LIN {X 0,Y 524.028,Z 204.208,A -85,B 0,C 180,E1 -4854.613,E2 -4854.613} C_VEL
LIN {X 0,Y 524.052,Z 204.202,A -85,B 0,C 180,E1 -4857.694,E2 -4857.694} C_VEL
LIN {X 0,Y 524.073,Z 204.206,A -85,B 0,C 180,E1 -4860.768,E2 -4860.768} C_VEL
LIN {X 0,Y 524.024,Z 204.211,A -85,B 0,C 180,E1 -4863.075,E2 -4863.075} C_VEL
LIN {X 0,Y 523.997,Z 204.21,A -85,B 0,C 180,E1 -4866.159,E2 -4866.159} C_VEL
LIN {X 0,Y 523.954,Z 204.219,A -85,B 0,C 180,E1 -4868.485,E2 -4868.485} C_VEL
LIN {X 0,Y 523.97,Z 204.212,A -85,B 0,C 180,E1 -4871.752,E2 -4871.752} C_VEL
LIN {X 0,Y 523.939,Z 204.219,A -85,B 0,C 180,E1 -4875.054,E2 -4875.054} C_VEL
LIN {X 0,Y 523.919,Z 204.219,A -85,B 0,C 180,E1 -4877.97,E2 -4877.97} C_VEL
LIN {X 0,Y 523.945,Z 204.222,A -85,B 0,C 180,E1 -4880.411,E2 -4880.411} C_VEL
LIN {X 0,Y 523.927,Z 204.221,A -85,B 0,C 180,E1 -4882.893,E2 -4882.893} C_VEL
LIN {X 0,Y 523.911,Z 204.219,A -85,B 0,C 180,E1 -4885.421,E2 -4885.421} C_VEL
LIN {X 0,Y 523.927,Z 204.221,A -85,B 0,C 180,E1 -4888.001,E2 -4888.001} C_VEL
LIN {X 0,Y 523.908,Z 204.222,A -85,B 0,C 180,E1 -4890.859,E2 -4890.859} C_VEL
LIN {X 0,Y 523.922,Z 204.22,A -85,B 0,C 180,E1 -4893.738,E2 -4893.738} C_VEL
LIN {X 0,Y 523.886,Z 204.229,A -85,B 0,C 180,E1 -4896.407,E2 -4896.407} C_VEL
LIN {X 0,Y 523.932,Z 204.217,A -85,B 0,C 180,E1 -4899.083,E2 -4899.083} C_VEL
LIN {X 0,Y 523.949,Z 204.215,A -85,B 0,C 180,E1 -4901.317,E2 -4901.317} C_VEL
LIN {X 0,Y 523.924,Z 204.219,A -85,B 0,C 180,E1 -4904.694,E2 -4904.694} C_VEL
LIN {X 0,Y 523.889,Z 204.222,A -85,B 0,C 180,E1 -4906.958,E2 -4906.958} C_VEL
LIN {X 0,Y 523.23,Z 204.308,A -85,B 0,C 180,E1 -4907.6,E2 -4907.6} C_VEL
LIN {X 0,Y 520.401,Z 204.663,A -85,B 0,C 180,E1 -4908.642,E2 -4908.642} C_VEL
LIN {X 0,Y 518.002,Z 204.964,A -85,B 0,C 180,E1 -4909.482,E2 -4909.482} C_VEL
LIN {X 0,Y 516.964,Z 205.091,A -85,B 0,C 180,E1 -4910.13,E2 -4910.13} C_VEL
LIN {X 0,Y 516.875,Z 205.099,A -85,B 0,C 180,E1 -4910.349,E2 -4910.349} C_VEL
LIN {X 0,Y 516.863,Z 205.099,A -85,B 0,C 180,E1 -4913.345,E2 -4913.345} C_VEL
LIN {X 0,Y 516.894,Z 205.098,A -85,B 0,C 180,E1 -4916.124,E2 -4916.124} C_VEL
LIN {X 0,Y 516.878,Z 205.095,A -85,B 0,C 180,E1 -4918.938,E2 -4918.938} C_VEL
LIN {X 0,Y 516.907,Z 205.098,A -85,B 0,C 180,E1 -4921.588,E2 -4921.588} C_VEL
LIN {X 0,Y 516.921,Z 205.092,A -85,B 0,C 180,E1 -4924.214,E2 -4924.214} C_VEL
LIN {X 0,Y 516.862,Z 205.097,A -85,B 0,C 180,E1 -4926.779,E2 -4926.779} C_VEL
LIN {X 0,Y 516.931,Z 205.096,A -85,B 0,C 180,E1 -4929.734,E2 -4929.734} C_VEL
LIN {X 0,Y 516.923,Z 205.09,A -85,B 0,C 180,E1 -4932.598,E2 -4932.598} C_VEL
LIN {X 0,Y 516.946,Z 205.09,A -85,B 0,C 180,E1 -4935.032,E2 -4935.032} C_VEL
LIN {X 0,Y 516.962,Z 205.085,A -85,B 0,C 180,E1 -4938.235,E2 -4938.235} C_VEL
LIN {X 0,Y 516.967,Z 205.093,A -85,B 0,C 180,E1 -4941.401,E2 -4941.401} C_VEL
LIN {X 0,Y 517,Z 205.083,A -85,B 0,C 180,E1 -4943.757,E2 -4943.757} C_VEL
LIN {X 0,Y 517.01,Z 205.082,A -85,B 0,C 180,E1 -4946.883,E2 -4946.883} C_VEL
LIN {X 0,Y 517.085,Z 205.07,A -85,B 0,C 180,E1 -4950,E2 -4950} C_VEL
LIN {X 0,Y 517.012,Z 205.088,A -85,B 0,C 180,E1 -4953.117,E2 -4953.117} C_VEL
LIN {X 0,Y 516.996,Z 205.081,A -85,B 0,C 180,E1 -4956.243,E2 -4956.243} C_VEL
LIN {X 0,Y 516.95,Z 205.09,A -85,B 0,C 180,E1 -4959.388,E2 -4959.388} C_VEL
LIN {X 0,Y 516.949,Z 205.087,A -85,B 0,C 180,E1 -4961.806,E2 -4961.806} C_VEL
LIN {X 0,Y 516.94,Z 205.093,A -85,B 0,C 180,E1 -4965.145,E2 -4965.145} C_VEL
LIN {X 0,Y 516.919,Z 205.091,A -85,B 0,C 180,E1 -4968.22,E2 -4968.22} C_VEL
LIN {X 0,Y 516.905,Z 205.099,A -85,B 0,C 180,E1 -4970.699,E2 -4970.699} C_VEL
LIN {X 0,Y 516.901,Z 205.093,A -85,B 0,C 180,E1 -4974.07,E2 -4974.07} C_VEL
LIN {X 0,Y 516.917,Z 205.1,A -85,B 0,C 180,E1 -4976.655,E2 -4976.655} C_VEL
LIN {X 0,Y 516.913,Z 205.095,A -85,B 0,C 180,E1 -4979.525,E2 -4979.525} C_VEL
LIN {X 0,Y 516.991,Z 205.141,A -85,B 0,C 180,E1 -4980.941,E2 -4980.941} C_VEL
LIN {X 0,Y 517.439,Z 210.279,A -85,B 0,C 180,E1 -4981.982,E2 -4981.982} C_VEL
LIN {X 0,Y 517.248,Z 224.094,A -85,B 0,C 180,E1 -4984.686,E2 -4984.686} C_VEL
LIN {X 0,Y 519.109,Z 235.104,A -85,B 0,C 180,E1 -4984.919,E2 -4984.919} C_VEL
LIN {X 0,Y 518.527,Z 331.623,A -85,B 0,C 180,E1 -4986.303,E2 -4986.303} C_VEL
LIN {X 0,Y 518.327,Z 345.145,A -85,B 0,C 180,E1 -4986.668,E2 -4986.668} C_VEL
LIN {X 0,Y 518.194,Z 357.087,A -85,B 0,C 180,E1 -4987.144,E2 -4987.144} C_VEL
LIN {X 0,Y 517.927,Z 368.274,A -85,B 0,C 180,E1 -4987.737,E2 -4987.737} C_VEL
LIN {X 0,Y 517.619,Z 379.34,A -85,B 0,C 180,E1 -4988.487,E2 -4988.487} C_VEL
LIN {X 0,Y 517.308,Z 390.499,A -85,B 0,C 180,E1 -4989.437,E2 -4989.437} C_VEL
LIN {X 0,Y 517.044,Z 399.867,A -85,B 0,C 180,E1 -4990.431,E2 -4990.431} C_VEL
LIN {X 0,Y 516.822,Z 408.68,A -85,B 0,C 180,E1 -4991.59,E2 -4991.59} C_VEL
LIN {X 0,Y 516.577,Z 416.392,A -85,B 0,C 180,E1 -4992.857,E2 -4992.857} C_VEL
LIN {X 0,Y 516.485,Z 422.702,A -85,B 0,C 180,E1 -4994.189,E2 -4994.189} C_VEL
LIN {X 0,Y 516.339,Z 427.576,A -85,B 0,C 180,E1 -4995.541,E2 -4995.541} C_VEL
LIN {X 0,Y 516.293,Z 430.487,A -85,B 0,C 180,E1 -4996.636,E2 -4996.636} C_VEL
LIN {X 0,Y 516.24,Z 433.161,A -85,B 0,C 180,E1 -4998.159,E2 -4998.159} C_VEL
LIN {X 0,Y 516.175,Z 434.262,A -85,B 0,C 180,E1 -4999.675,E2 -4999.675} C_VEL
LIN {X 0,Y 516.192,Z 433.883,A -85,B 0,C 180,E1 -5001.223,E2 -5001.223} C_VEL
LIN {X 0,Y 516.191,Z 432.79,A -85,B 0,C 180,E1 -5002.217,E2 -5002.217} C_VEL
LIN {X 0,Y 516.28,Z 430.595,A -85,B 0,C 180,E1 -5003.424,E2 -5003.424} C_VEL
LIN {X 0,Y 516.358,Z 427.029,A -85,B 0,C 180,E1 -5004.741,E2 -5004.741} C_VEL
LIN {X 0,Y 516.425,Z 421.942,A -85,B 0,C 180,E1 -5006.104,E2 -5006.104} C_VEL
LIN {X 0,Y 516.6,Z 416.145,A -85,B 0,C 180,E1 -5007.295,E2 -5007.295} C_VEL
LIN {X 0,Y 516.793,Z 409.28,A -85,B 0,C 180,E1 -5008.428,E2 -5008.428} C_VEL
LIN {X 0,Y 517.047,Z 400.626,A -85,B 0,C 180,E1 -5009.581,E2 -5009.581} C_VEL
LIN {X 0,Y 517.308,Z 391.616,A -85,B 0,C 180,E1 -5010.557,E2 -5010.557} C_VEL
LIN {X 0,Y 517.528,Z 382.117,A -85,B 0,C 180,E1 -5011.4,E2 -5011.4} C_VEL
LIN {X 0,Y 517.83,Z 371.744,A -85,B 0,C 180,E1 -5012.145,E2 -5012.145} C_VEL
LIN {X 0,Y 518.169,Z 359.936,A -85,B 0,C 180,E1 -5012.813,E2 -5012.813} C_VEL
LIN {X 0,Y 518.374,Z 348.271,A -85,B 0,C 180,E1 -5013.314,E2 -5013.314} C_VEL
LIN {X 0,Y 518.512,Z 335.514,A -85,B 0,C 180,E1 -5013.702,E2 -5013.702} C_VEL
LIN {X 0,Y 518.61,Z 319.67,A -85,B 0,C 180,E1 -5013.977,E2 -5013.977} C_VEL
LIN {X 0,Y 519.05,Z 233.514,A -85,B 0,C 180,E1 -5015.201,E2 -5015.201} C_VEL
LIN {X 0,Y 517.236,Z 223.957,A -85,B 0,C 180,E1 -5015.41,E2 -5015.41} C_VEL
LIN {X 0,Y 517.224,Z 207.844,A -85,B 0,C 180,E1 -5018.268,E2 -5018.268} C_VEL
LIN {X 0,Y 516.917,Z 205.098,A -85,B 0,C 180,E1 -5018.778,E2 -5018.778} C_VEL
LIN {X 0,Y 516.879,Z 205.098,A -85,B 0,C 180,E1 -5022.117,E2 -5022.117} C_VEL
LIN {X 0,Y 516.897,Z 205.1,A -85,B 0,C 180,E1 -5025.029,E2 -5025.029} C_VEL
LIN {X 0,Y 516.951,Z 205.09,A -85,B 0,C 180,E1 -5028.234,E2 -5028.234} C_VEL
LIN {X 0,Y 516.92,Z 205.098,A -85,B 0,C 180,E1 -5031.399,E2 -5031.399} C_VEL
LIN {X 0,Y 516.966,Z 205.088,A -85,B 0,C 180,E1 -5033.757,E2 -5033.757} C_VEL
LIN {X 0,Y 516.966,Z 205.091,A -85,B 0,C 180,E1 -5036.883,E2 -5036.883} C_VEL
LIN {X 0,Y 517.024,Z 205.079,A -85,B 0,C 180,E1 -5040,E2 -5040} C_VEL
LIN {X 0,Y 516.964,Z 205.092,A -85,B 0,C 180,E1 -5043.118,E2 -5043.118} C_VEL
LIN {X 0,Y 516.947,Z 205.087,A -85,B 0,C 180,E1 -5046.244,E2 -5046.244} C_VEL
LIN {X 0,Y 516.907,Z 205.095,A -85,B 0,C 180,E1 -5049.39,E2 -5049.39} C_VEL
LIN {X 0,Y 516.931,Z 205.088,A -85,B 0,C 180,E1 -5051.826,E2 -5051.826} C_VEL
LIN {X 0,Y 516.891,Z 205.098,A -85,B 0,C 180,E1 -5055.147,E2 -5055.147} C_VEL
LIN {X 0,Y 516.881,Z 205.097,A -85,B 0,C 180,E1 -5058.224,E2 -5058.224} C_VEL
LIN {X 0,Y 516.867,Z 205.104,A -85,B 0,C 180,E1 -5060.704,E2 -5060.704} C_VEL
LIN {X 0,Y 516.844,Z 205.099,A -85,B 0,C 180,E1 -5063.225,E2 -5063.225} C_VEL
LIN {X 0,Y 516.9,Z 205.097,A -85,B 0,C 180,E1 -5066.199,E2 -5066.199} C_VEL
LIN {X 0,Y 516.881,Z 205.094,A -85,B 0,C 180,E1 -5069.307,E2 -5069.307} C_VEL
LIN {X 0,Y 516.861,Z 205.104,A -85,B 0,C 180,E1 -5072.547,E2 -5072.547} C_VEL
LIN {X 0,Y 516.846,Z 205.098,A -85,B 0,C 180,E1 -5075.335,E2 -5075.335} C_VEL
LIN {X 0,Y 516.847,Z 205.103,A -85,B 0,C 180,E1 -5077.946,E2 -5077.946} C_VEL
LIN {X 0,Y 516.854,Z 205.101,A -85,B 0,C 180,E1 -5080.745,E2 -5080.745} C_VEL
LIN {X 0,Y 516.855,Z 205.099,A -85,B 0,C 180,E1 -5082.835,E2 -5082.835} C_VEL
LIN {X 0,Y 516.869,Z 205.097,A -85,B 0,C 180,E1 -5085.01,E2 -5085.01} C_VEL
LIN {X 0,Y 516.894,Z 205.099,A -85,B 0,C 180,E1 -5088.402,E2 -5088.402} C_VEL
LIN {X 0,Y 516.86,Z 205.099,A -85,B 0,C 180,E1 -5091.287,E2 -5091.287} C_VEL
LIN {X 0,Y 516.871,Z 205.103,A -85,B 0,C 180,E1 -5094.224,E2 -5094.224} C_VEL
LIN {X 0,Y 516.88,Z 205.097,A -85,B 0,C 180,E1 -5097.056,E2 -5097.056} C_VEL
LIN {X 0,Y 516.88,Z 205.104,A -85,B 0,C 180,E1 -5099.799,E2 -5099.799} C_VEL
LIN {X 0,Y 516.915,Z 205.096,A -85,B 0,C 180,E1 -5102.47,E2 -5102.47} C_VEL
LIN {X 0,Y 516.957,Z 205.158,A -85,B 0,C 180,E1 -5105.114,E2 -5105.114} C_VEL
LIN {X 0,Y 518.311,Z 213.375,A -85,B 0,C 180,E1 -5106.424,E2 -5106.424} C_VEL
LIN {X 0,Y 517.948,Z 232.817,A -85,B 0,C 180,E1 -5109.344,E2 -5109.344} C_VEL
LIN {X 0,Y 517.523,Z 253.595,A -85,B 0,C 180,E1 -5112.442,E2 -5112.442} C_VEL
LIN {X 0,Y 517.213,Z 268.372,A -85,B 0,C 180,E1 -5114.627,E2 -5114.627} C_VEL
LIN {X 0,Y 519.009,Z 281.849,A -85,B 0,C 180,E1 -5114.879,E2 -5114.879} C_VEL
LIN {X 0,Y 518.499,Z 377.861,A -85,B 0,C 180,E1 -5116.255,E2 -5116.255} C_VEL
LIN {X 0,Y 518.253,Z 391.659,A -85,B 0,C 180,E1 -5116.623,E2 -5116.623} C_VEL
LIN {X 0,Y 517.973,Z 404.074,A -85,B 0,C 180,E1 -5117.114,E2 -5117.114} C_VEL
LIN {X 0,Y 517.695,Z 416.837,A -85,B 0,C 180,E1 -5117.808,E2 -5117.808} C_VEL
LIN {X 0,Y 517.391,Z 428.749,A -85,B 0,C 180,E1 -5118.642,E2 -5118.642} C_VEL
LIN {X 0,Y 517.132,Z 437.799,A -85,B 0,C 180,E1 -5119.429,E2 -5119.429} C_VEL
LIN {X 0,Y 516.852,Z 447.086,A -85,B 0,C 180,E1 -5120.412,E2 -5120.412} C_VEL
LIN {X 0,Y 516.635,Z 456.126,A -85,B 0,C 180,E1 -5121.592,E2 -5121.592} C_VEL
LIN {X 0,Y 516.502,Z 463.409,A -85,B 0,C 180,E1 -5122.77,E2 -5122.77} C_VEL
LIN {X 0,Y 516.383,Z 468.318,A -85,B 0,C 180,E1 -5123.75,E2 -5123.75} C_VEL
LIN {X 0,Y 516.312,Z 473.094,A -85,B 0,C 180,E1 -5124.924,E2 -5124.924} C_VEL
LIN {X 0,Y 516.37,Z 476.747,A -85,B 0,C 180,E1 -5126.098,E2 -5126.098} C_VEL
LIN {X 0,Y 516.282,Z 478.629,A -85,B 0,C 180,E1 -5126.879,E2 -5126.879} C_VEL
LIN {X 0,Y 516.261,Z 480.041,A -85,B 0,C 180,E1 -5127.66,E2 -5127.66} C_VEL
LIN {X 0,Y 516.167,Z 481.664,A -85,B 0,C 180,E1 -5129.22,E2 -5129.22} C_VEL
LIN {X 0,Y 516.167,Z 481.887,A -85,B 0,C 180,E1 -5130,E2 -5130} C_VEL
LIN {X 0,Y 516.192,Z 481.066,A -85,B 0,C 180,E1 -5131.56,E2 -5131.56} C_VEL
LIN {X 0,Y 516.261,Z 480.07,A -85,B 0,C 180,E1 -5132.34,E2 -5132.34} C_VEL
LIN {X 0,Y 516.282,Z 478.667,A -85,B 0,C 180,E1 -5133.121,E2 -5133.121} C_VEL
LIN {X 0,Y 516.311,Z 475.715,A -85,B 0,C 180,E1 -5134.293,E2 -5134.293} C_VEL
LIN {X 0,Y 516.368,Z 471.715,A -85,B 0,C 180,E1 -5135.466,E2 -5135.466} C_VEL
LIN {X 0,Y 516.439,Z 465.782,A -85,B 0,C 180,E1 -5136.794,E2 -5136.794} C_VEL
LIN {X 0,Y 516.592,Z 458.83,A -85,B 0,C 180,E1 -5138.015,E2 -5138.015} C_VEL
LIN {X 0,Y 516.77,Z 450.482,A -85,B 0,C 180,E1 -5139.194,E2 -5139.194} C_VEL
LIN {X 0,Y 516.971,Z 441.909,A -85,B 0,C 180,E1 -5140.178,E2 -5140.178} C_VEL
LIN {X 0,Y 517.33,Z 431.327,A -85,B 0,C 180,E1 -5141.161,E2 -5141.161} C_VEL
LIN {X 0,Y 517.674,Z 420.056,A -85,B 0,C 180,E1 -5142.002,E2 -5142.002} C_VEL
LIN {X 0,Y 517.9,Z 409.336,A -85,B 0,C 180,E1 -5142.638,E2 -5142.638} C_VEL
LIN {X 0,Y 518.141,Z 397.418,A -85,B 0,C 180,E1 -5143.18,E2 -5143.18} C_VEL
LIN {X 0,Y 518.418,Z 383.678,A -85,B 0,C 180,E1 -5143.622,E2 -5143.622} C_VEL
LIN {X 0,Y 518.627,Z 371.26,A -85,B 0,C 180,E1 -5143.866,E2 -5143.866} C_VEL
LIN {X 0,Y 518.844,Z 279.698,A -85,B 0,C 180,E1 -5145.162,E2 -5145.162} C_VEL
LIN {X 0,Y 517.252,Z 268.853,A -85,B 0,C 180,E1 -5145.371,E2 -5145.371} C_VEL
LIN {X 0,Y 517.694,Z 248.791,A -85,B 0,C 180,E1 -5148.397,E2 -5148.397} C_VEL
LIN {X 0,Y 518.264,Z 228.616,A -85,B 0,C 180,E1 -5151.475,E2 -5151.475} C_VEL
LIN {X 0,Y 518.602,Z 213.817,A -85,B 0,C 180,E1 -5153.773,E2 -5153.773} C_VEL
LIN {X 0,Y 516.949,Z 205.092,A -85,B 0,C 180,E1 -5155.246,E2 -5155.246} C_VEL
LIN {X 0,Y 516.904,Z 205.099,A -85,B 0,C 180,E1 -5158.413,E2 -5158.413} C_VEL
LIN {X 0,Y 516.876,Z 205.097,A -85,B 0,C 180,E1 -5161.106,E2 -5161.106} C_VEL
LIN {X 0,Y 516.895,Z 205.102,A -85,B 0,C 180,E1 -5163.963,E2 -5163.963} C_VEL
LIN {X 0,Y 516.864,Z 205.097,A -85,B 0,C 180,E1 -5166.742,E2 -5166.742} C_VEL
LIN {X 0,Y 516.86,Z 205.104,A -85,B 0,C 180,E1 -5169.718,E2 -5169.718} C_VEL
LIN {X 0,Y 516.891,Z 205.102,A -85,B 0,C 180,E1 -5171.771,E2 -5171.771} C_VEL
LIN {X 0,Y 516.896,Z 205.093,A -85,B 0,C 180,E1 -5175.007,E2 -5175.007} C_VEL
LIN {X 0,Y 516.886,Z 205.095,A -85,B 0,C 180,E1 -5178.395,E2 -5178.395} C_VEL
LIN {X 0,Y 516.847,Z 205.103,A -85,B 0,C 180,E1 -5181.281,E2 -5181.281} C_VEL
LIN {X 0,Y 516.855,Z 205.1,A -85,B 0,C 180,E1 -5184.218,E2 -5184.218} C_VEL
LIN {X 0,Y 516.859,Z 205.1,A -85,B 0,C 180,E1 -5187.05,E2 -5187.05} C_VEL
LIN {X 0,Y 516.85,Z 205.104,A -85,B 0,C 180,E1 -5189.793,E2 -5189.793} C_VEL
LIN {X 0,Y 516.886,Z 205.094,A -85,B 0,C 180,E1 -5192.465,E2 -5192.465} C_VEL
LIN {X 0,Y 516.867,Z 205.101,A -85,B 0,C 180,E1 -5195.069,E2 -5195.069} C_VEL
LIN {X 0,Y 516.866,Z 205.102,A -85,B 0,C 180,E1 -5197.621,E2 -5197.621} C_VEL
LIN {X 0,Y 516.883,Z 205.095,A -85,B 0,C 180,E1 -5200.128,E2 -5200.128} C_VEL
LIN {X 0,Y 516.891,Z 205.095,A -85,B 0,C 180,E1 -5202.595,E2 -5202.595} C_VEL
LIN {X 0,Y 516.888,Z 205.1,A -85,B 0,C 180,E1 -5205.028,E2 -5205.028} C_VEL
LIN {X 0,Y 516.951,Z 205.086,A -85,B 0,C 180,E1 -5208.233,E2 -5208.233} C_VEL
LIN {X 0,Y 516.917,Z 205.095,A -85,B 0,C 180,E1 -5211.399,E2 -5211.399} C_VEL
LIN {X 0,Y 516.946,Z 205.088,A -85,B 0,C 180,E1 -5213.756,E2 -5213.756} C_VEL
LIN {X 0,Y 516.963,Z 205.092,A -85,B 0,C 180,E1 -5216.882,E2 -5216.882} C_VEL
LIN {X 0,Y 517.023,Z 205.077,A -85,B 0,C 180,E1 -5220,E2 -5220} C_VEL
LIN {X 0,Y 516.965,Z 205.09,A -85,B 0,C 180,E1 -5223.117,E2 -5223.117} C_VEL
LIN {X 0,Y 516.965,Z 205.086,A -85,B 0,C 180,E1 -5226.243,E2 -5226.243} C_VEL
LIN {X 0,Y 516.919,Z 205.097,A -85,B 0,C 180,E1 -5228.601,E2 -5228.601} C_VEL
LIN {X 0,Y 516.929,Z 205.089,A -85,B 0,C 180,E1 -5231.825,E2 -5231.825} C_VEL
LIN {X 0,Y 516.892,Z 205.096,A -85,B 0,C 180,E1 -5235.148,E2 -5235.148} C_VEL
LIN {X 0,Y 516.879,Z 205.099,A -85,B 0,C 180,E1 -5238.224,E2 -5238.224} C_VEL
LIN {X 0,Y 516.884,Z 205.101,A -85,B 0,C 180,E1 -5240.702,E2 -5240.702} C_VEL
LIN {X 0,Y 516.867,Z 205.097,A -85,B 0,C 180,E1 -5243.223,E2 -5243.223} C_VEL
LIN {X 0,Y 516.898,Z 205.098,A -85,B 0,C 180,E1 -5246.199,E2 -5246.199} C_VEL
LIN {X 0,Y 516.898,Z 205.093,A -85,B 0,C 180,E1 -5249.306,E2 -5249.306} C_VEL
LIN {X 0,Y 516.859,Z 205.103,A -85,B 0,C 180,E1 -5252.547,E2 -5252.547} C_VEL
LIN {X 0,Y 516.844,Z 205.1,A -85,B 0,C 180,E1 -5255.335,E2 -5255.335} C_VEL
LIN {X 0,Y 516.846,Z 205.104,A -85,B 0,C 180,E1 -5257.946,E2 -5257.946} C_VEL
LIN {X 0,Y 516.883,Z 205.096,A -85,B 0,C 180,E1 -5260.741,E2 -5260.741} C_VEL
LIN {X 0,Y 516.851,Z 205.105,A -85,B 0,C 180,E1 -5263.906,E2 -5263.906} C_VEL
LIN {X 0,Y 516.853,Z 205.107,A -85,B 0,C 180,E1 -5266.11,E2 -5266.11} C_VEL
LIN {X 0,Y 516.886,Z 205.095,A -85,B 0,C 180,E1 -5269.264,E2 -5269.264} C_VEL
LIN {X 0,Y 516.875,Z 205.099,A -85,B 0,C 180,E1 -5270.349,E2 -5270.349} C_VEL
LIN {X 0,Y 516.197,Z 205.181,A -85,B 0,C 180,E1 -5270.999,E2 -5270.999} C_VEL
LIN {X 0,Y 513.342,Z 205.543,A -85,B 0,C 180,E1 -5272.055,E2 -5272.055} C_VEL
LIN {X 0,Y 510.933,Z 205.845,A -85,B 0,C 180,E1 -5272.905,E2 -5272.905} C_VEL
LIN {X 0,Y 509.895,Z 205.971,A -85,B 0,C 180,E1 -5273.562,E2 -5273.562} C_VEL
LIN {X 0,Y 509.808,Z 205.98,A -85,B 0,C 180,E1 -5273.784,E2 -5273.784} C_VEL
LIN {X 0,Y 509.845,Z 205.972,A -85,B 0,C 180,E1 -5276.542,E2 -5276.542} C_VEL
LIN {X 0,Y 509.834,Z 205.976,A -85,B 0,C 180,E1 -5279.337,E2 -5279.337} C_VEL
LIN {X 0,Y 509.881,Z 205.971,A -85,B 0,C 180,E1 -5282.057,E2 -5282.057} C_VEL
LIN {X 0,Y 509.867,Z 205.969,A -85,B 0,C 180,E1 -5284.707,E2 -5284.707} C_VEL
LIN {X 0,Y 509.827,Z 205.98,A -85,B 0,C 180,E1 -5287.457,E2 -5287.457} C_VEL
LIN {X 0,Y 509.909,Z 205.969,A -85,B 0,C 180,E1 -5289.847,E2 -5289.847} C_VEL
LIN {X 0,Y 509.879,Z 205.971,A -85,B 0,C 180,E1 -5293.177,E2 -5293.177} C_VEL
LIN {X 0,Y 509.868,Z 205.975,A -85,B 0,C 180,E1 -5295.636,E2 -5295.636} C_VEL
LIN {X 0,Y 509.91,Z 205.965,A -85,B 0,C 180,E1 -5298.876,E2 -5298.876} C_VEL
LIN {X 0,Y 509.949,Z 205.959,A -85,B 0,C 180,E1 -5302.079,E2 -5302.079} C_VEL
LIN {X 0,Y 509.978,Z 205.955,A -85,B 0,C 180,E1 -5304.465,E2 -5304.465} C_VEL
LIN {X 0,Y 510.055,Z 205.949,A -85,B 0,C 180,E1 -5307.631,E2 -5307.631} C_VEL
LIN {X 0,Y 510.062,Z 205.948,A -85,B 0,C 180,E1 -5310.789,E2 -5310.789} C_VEL
LIN {X 0,Y 509.954,Z 205.967,A -85,B 0,C 180,E1 -5313.16,E2 -5313.16} C_VEL
LIN {X 0,Y 509.943,Z 205.96,A -85,B 0,C 180,E1 -5316.329,E2 -5316.329} C_VEL
LIN {X 0,Y 509.913,Z 205.967,A -85,B 0,C 180,E1 -5318.719,E2 -5318.719} C_VEL
LIN {X 0,Y 509.901,Z 205.964,A -85,B 0,C 180,E1 -5321.93,E2 -5321.93} C_VEL
LIN {X 0,Y 509.889,Z 205.97,A -85,B 0,C 180,E1 -5325.24,E2 -5325.24} C_VEL
LIN {X 0,Y 509.883,Z 205.967,A -85,B 0,C 180,E1 -5327.999,E2 -5327.999} C_VEL
LIN {X 0,Y 509.843,Z 205.978,A -85,B 0,C 180,E1 -5331,E2 -5331} C_VEL
LIN {X 0,Y 509.827,Z 205.974,A -85,B 0,C 180,E1 -5333.561,E2 -5333.561} C_VEL
LIN {X 0,Y 509.902,Z 205.97,A -85,B 0,C 180,E1 -5336.377,E2 -5336.377} C_VEL
LIN {X 0,Y 509.872,Z 205.976,A -85,B 0,C 180,E1 -5338.841,E2 -5338.841} C_VEL
LIN {X 0,Y 509.958,Z 205.983,A -85,B 0,C 180,E1 -5340.81,E2 -5340.81} C_VEL
LIN {X 0,Y 510.45,Z 210.705,A -85,B 0,C 180,E1 -5341.775,E2 -5341.775} C_VEL
LIN {X 0,Y 510.23,Z 224.338,A -85,B 0,C 180,E1 -5344.47,E2 -5344.47} C_VEL
LIN {X 0,Y 512.23,Z 234.881,A -85,B 0,C 180,E1 -5344.704,E2 -5344.704} C_VEL
LIN {X 0,Y 511.675,Z 330.813,A -85,B 0,C 180,E1 -5346.097,E2 -5346.097} C_VEL
LIN {X 0,Y 511.437,Z 344.08,A -85,B 0,C 180,E1 -5346.445,E2 -5346.445} C_VEL
LIN {X 0,Y 511.286,Z 357.191,A -85,B 0,C 180,E1 -5346.964,E2 -5346.964} C_VEL
LIN {X 0,Y 510.973,Z 369.148,A -85,B 0,C 180,E1 -5347.609,E2 -5347.609} C_VEL
LIN {X 0,Y 510.631,Z 380.814,A -85,B 0,C 180,E1 -5348.424,E2 -5348.424} C_VEL
LIN {X 0,Y 510.313,Z 390.903,A -85,B 0,C 180,E1 -5349.304,E2 -5349.304} C_VEL
LIN {X 0,Y 510.028,Z 400.624,A -85,B 0,C 180,E1 -5350.359,E2 -5350.359} C_VEL
LIN {X 0,Y 509.805,Z 408.629,A -85,B 0,C 180,E1 -5351.425,E2 -5351.425} C_VEL
LIN {X 0,Y 509.538,Z 415.352,A -85,B 0,C 180,E1 -5352.514,E2 -5352.514} C_VEL
LIN {X 0,Y 509.406,Z 422.088,A -85,B 0,C 180,E1 -5353.885,E2 -5353.885} C_VEL
LIN {X 0,Y 509.291,Z 427.23,A -85,B 0,C 180,E1 -5355.27,E2 -5355.27} C_VEL
LIN {X 0,Y 509.234,Z 430.296,A -85,B 0,C 180,E1 -5356.366,E2 -5356.366} C_VEL
LIN {X 0,Y 509.164,Z 432.48,A -85,B 0,C 180,E1 -5357.442,E2 -5357.442} C_VEL
LIN {X 0,Y 509.146,Z 433.872,A -85,B 0,C 180,E1 -5358.504,E2 -5358.504} C_VEL
LIN {X 0,Y 509.105,Z 434.56,A -85,B 0,C 180,E1 -5359.548,E2 -5359.548} C_VEL
LIN {X 0,Y 509.129,Z 434.553,A -85,B 0,C 180,E1 -5360.618,E2 -5360.618} C_VEL
LIN {X 0,Y 509.098,Z 433.597,A -85,B 0,C 180,E1 -5361.886,E2 -5361.886} C_VEL
LIN {X 0,Y 509.169,Z 431.562,A -85,B 0,C 180,E1 -5363.176,E2 -5363.176} C_VEL
LIN {X 0,Y 509.267,Z 428.061,A -85,B 0,C 180,E1 -5364.577,E2 -5364.577} C_VEL
LIN {X 0,Y 509.333,Z 423.536,A -85,B 0,C 180,E1 -5365.875,E2 -5365.875} C_VEL
LIN {X 0,Y 509.546,Z 417.111,A -85,B 0,C 180,E1 -5367.273,E2 -5367.273} C_VEL
LIN {X 0,Y 509.738,Z 410.51,A -85,B 0,C 180,E1 -5368.404,E2 -5368.404} C_VEL
LIN {X 0,Y 510.004,Z 402.045,A -85,B 0,C 180,E1 -5369.574,E2 -5369.574} C_VEL
LIN {X 0,Y 510.314,Z 392.712,A -85,B 0,C 180,E1 -5370.619,E2 -5370.619} C_VEL
LIN {X 0,Y 510.566,Z 383.025,A -85,B 0,C 180,E1 -5371.504,E2 -5371.504} C_VEL
LIN {X 0,Y 510.909,Z 371.564,A -85,B 0,C 180,E1 -5372.338,E2 -5372.338} C_VEL
LIN {X 0,Y 511.224,Z 359.501,A -85,B 0,C 180,E1 -5373.021,E2 -5373.021} C_VEL
LIN {X 0,Y 511.493,Z 346.514,A -85,B 0,C 180,E1 -5373.566,E2 -5373.566} C_VEL
LIN {X 0,Y 511.642,Z 333.326,A -85,B 0,C 180,E1 -5373.938,E2 -5373.938} C_VEL
LIN {X 0,Y 511.818,Z 308.174,A -85,B 0,C 180,E1 -5374.331,E2 -5374.331} C_VEL
LIN {X 0,Y 512.249,Z 234.752,A -85,B 0,C 180,E1 -5375.393,E2 -5375.393} C_VEL
LIN {X 0,Y 510.249,Z 224.241,A -85,B 0,C 180,E1 -5375.621,E2 -5375.621} C_VEL
LIN {X 0,Y 510.235,Z 208.761,A -85,B 0,C 180,E1 -5378.38,E2 -5378.38} C_VEL
LIN {X 0,Y 509.881,Z 205.975,A -85,B 0,C 180,E1 -5378.894,E2 -5378.894} C_VEL
LIN {X 0,Y 509.858,Z 205.972,A -85,B 0,C 180,E1 -5382.347,E2 -5382.347} C_VEL
LIN {X 0,Y 509.824,Z 205.983,A -85,B 0,C 180,E1 -5385.633,E2 -5385.633} C_VEL
LIN {X 0,Y 509.891,Z 205.97,A -85,B 0,C 180,E1 -5388.1,E2 -5388.1} C_VEL
LIN {X 0,Y 509.867,Z 205.978,A -85,B 0,C 180,E1 -5391.279,E2 -5391.279} C_VEL
LIN {X 0,Y 509.937,Z 205.964,A -85,B 0,C 180,E1 -5393.67,E2 -5393.67} C_VEL
LIN {X 0,Y 509.908,Z 205.969,A -85,B 0,C 180,E1 -5396.84,E2 -5396.84} C_VEL
LIN {X 0,Y 510.014,Z 205.959,A -85,B 0,C 180,E1 -5399.211,E2 -5399.211} C_VEL
LIN {X 0,Y 509.882,Z 205.97,A -85,B 0,C 180,E1 -5401.58,E2 -5401.58} C_VEL
LIN {X 0,Y 509.906,Z 205.971,A -85,B 0,C 180,E1 -5403.161,E2 -5403.161} C_VEL
LIN {X 0,Y 509.898,Z 205.965,A -85,B 0,C 180,E1 -5406.331,E2 -5406.331} C_VEL
LIN {X 0,Y 509.865,Z 205.975,A -85,B 0,C 180,E1 -5408.721,E2 -5408.721} C_VEL
LIN {X 0,Y 509.9,Z 205.964,A -85,B 0,C 180,E1 -5411.932,E2 -5411.932} C_VEL
LIN {X 0,Y 509.844,Z 205.975,A -85,B 0,C 180,E1 -5415.244,E2 -5415.244} C_VEL
LIN {X 0,Y 509.84,Z 205.972,A -85,B 0,C 180,E1 -5418.003,E2 -5418.003} C_VEL
LIN {X 0,Y 509.809,Z 205.981,A -85,B 0,C 180,E1 -5421.004,E2 -5421.004} C_VEL
LIN {X 0,Y 509.804,Z 205.975,A -85,B 0,C 180,E1 -5423.565,E2 -5423.565} C_VEL
LIN {X 0,Y 509.869,Z 205.975,A -85,B 0,C 180,E1 -5426.381,E2 -5426.381} C_VEL
LIN {X 0,Y 509.836,Z 205.976,A -85,B 0,C 180,E1 -5428.847,E2 -5428.847} C_VEL
LIN {X 0,Y 509.785,Z 205.98,A -85,B 0,C 180,E1 -5431.593,E2 -5431.593} C_VEL
LIN {X 0,Y 509.816,Z 205.983,A -85,B 0,C 180,E1 -5434.416,E2 -5434.416} C_VEL
LIN {X 0,Y 509.785,Z 205.98,A -85,B 0,C 180,E1 -5437.344,E2 -5437.344} C_VEL
LIN {X 0,Y 509.807,Z 205.983,A -85,B 0,C 180,E1 -5440.386,E2 -5440.386} C_VEL
LIN {X 0,Y 509.795,Z 205.977,A -85,B 0,C 180,E1 -5443.066,E2 -5443.066} C_VEL
LIN {X 0,Y 509.797,Z 205.981,A -85,B 0,C 180,E1 -5445.797,E2 -5445.797} C_VEL
LIN {X 0,Y 509.836,Z 205.976,A -85,B 0,C 180,E1 -5448.578,E2 -5448.578} C_VEL
LIN {X 0,Y 509.831,Z 205.979,A -85,B 0,C 180,E1 -5451.79,E2 -5451.79} C_VEL
LIN {X 0,Y 509.827,Z 205.976,A -85,B 0,C 180,E1 -5454.626,E2 -5454.626} C_VEL
LIN {X 0,Y 509.847,Z 205.976,A -85,B 0,C 180,E1 -5457.484,E2 -5457.484} C_VEL
LIN {X 0,Y 509.848,Z 205.979,A -85,B 0,C 180,E1 -5460.277,E2 -5460.277} C_VEL
LIN {X 0,Y 509.873,Z 205.972,A -85,B 0,C 180,E1 -5462.947,E2 -5462.947} C_VEL
LIN {X 0,Y 509.909,Z 206.106,A -85,B 0,C 180,E1 -5464.963,E2 -5464.963} C_VEL
LIN {X 0,Y 511.329,Z 214.333,A -85,B 0,C 180,E1 -5466.298,E2 -5466.298} C_VEL
LIN {X 0,Y 511.005,Z 232.375,A -85,B 0,C 180,E1 -5469.05,E2 -5469.05} C_VEL
LIN {X 0,Y 510.502,Z 254.403,A -85,B 0,C 180,E1 -5472.372,E2 -5472.372} C_VEL
LIN {X 0,Y 510.216,Z 267.995,A -85,B 0,C 180,E1 -5474.409,E2 -5474.409} C_VEL
LIN {X 0,Y 512.149,Z 282.754,A -85,B 0,C 180,E1 -5474.69,E2 -5474.69} C_VEL
LIN {X 0,Y 511.617,Z 377.203,A -85,B 0,C 180,E1 -5476.066,E2 -5476.066} C_VEL
LIN {X 0,Y 511.331,Z 390.33,A -85,B 0,C 180,E1 -5476.413,E2 -5476.413} C_VEL
LIN {X 0,Y 511.033,Z 403.576,A -85,B 0,C 180,E1 -5476.936,E2 -5476.936} C_VEL
LIN {X 0,Y 510.753,Z 416.122,A -85,B 0,C 180,E1 -5477.623,E2 -5477.623} C_VEL
LIN {X 0,Y 510.396,Z 427.015,A -85,B 0,C 180,E1 -5478.383,E2 -5478.383} C_VEL
LIN {X 0,Y 510.126,Z 437.385,A -85,B 0,C 180,E1 -5479.282,E2 -5479.282} C_VEL
LIN {X 0,Y 509.82,Z 446.69,A -85,B 0,C 180,E1 -5480.279,E2 -5480.279} C_VEL
LIN {X 0,Y 509.586,Z 455.746,A -85,B 0,C 180,E1 -5481.475,E2 -5481.475} C_VEL
LIN {X 0,Y 509.424,Z 463.04,A -85,B 0,C 180,E1 -5482.669,E2 -5482.669} C_VEL
LIN {X 0,Y 509.308,Z 467.96,A -85,B 0,C 180,E1 -5483.663,E2 -5483.663} C_VEL
LIN {X 0,Y 509.241,Z 472.745,A -85,B 0,C 180,E1 -5484.854,E2 -5484.854} C_VEL
LIN {X 0,Y 509.275,Z 476.406,A -85,B 0,C 180,E1 -5486.044,E2 -5486.044} C_VEL
LIN {X 0,Y 509.201,Z 478.292,A -85,B 0,C 180,E1 -5486.835,E2 -5486.835} C_VEL
LIN {X 0,Y 509.19,Z 479.708,A -85,B 0,C 180,E1 -5487.627,E2 -5487.627} C_VEL
LIN {X 0,Y 509.08,Z 481.336,A -85,B 0,C 180,E1 -5489.209,E2 -5489.209} C_VEL
LIN {X 0,Y 509.078,Z 481.561,A -85,B 0,C 180,E1 -5490,E2 -5490} C_VEL
LIN {X 0,Y 509.112,Z 480.741,A -85,B 0,C 180,E1 -5491.582,E2 -5491.582} C_VEL
LIN {X 0,Y 509.19,Z 479.746,A -85,B 0,C 180,E1 -5492.373,E2 -5492.373} C_VEL
LIN {X 0,Y 509.2,Z 478.34,A -85,B 0,C 180,E1 -5493.164,E2 -5493.164} C_VEL
LIN {X 0,Y 509.204,Z 475.384,A -85,B 0,C 180,E1 -5494.353,E2 -5494.353} C_VEL
LIN {X 0,Y 509.283,Z 471.381,A -85,B 0,C 180,E1 -5495.543,E2 -5495.543} C_VEL
LIN {X 0,Y 509.35,Z 465.67,A -85,B 0,C 180,E1 -5496.844,E2 -5496.844} C_VEL
LIN {X 0,Y 509.513,Z 458.48,A -85,B 0,C 180,E1 -5498.127,E2 -5498.127} C_VEL
LIN {X 0,Y 509.717,Z 450.124,A -85,B 0,C 180,E1 -5499.322,E2 -5499.322} C_VEL
LIN {X 0,Y 509.947,Z 441.537,A -85,B 0,C 180,E1 -5500.32,E2 -5500.32} C_VEL
LIN {X 0,Y 510.341,Z 430.943,A -85,B 0,C 180,E1 -5501.316,E2 -5501.316} C_VEL
LIN {X 0,Y 510.666,Z 419.653,A -85,B 0,C 180,E1 -5502.17,E2 -5502.17} C_VEL
LIN {X 0,Y 510.936,Z 408.907,A -85,B 0,C 180,E1 -5502.813,E2 -5502.813} C_VEL
LIN {X 0,Y 511.188,Z 396.947,A -85,B 0,C 180,E1 -5503.363,E2 -5503.363} C_VEL
LIN {X 0,Y 511.531,Z 383.157,A -85,B 0,C 180,E1 -5503.809,E2 -5503.809} C_VEL
LIN {X 0,Y 511.73,Z 370.554,A -85,B 0,C 180,E1 -5504.057,E2 -5504.057} C_VEL
LIN {X 0,Y 511.994,Z 280.449,A -85,B 0,C 180,E1 -5505.354,E2 -5505.354} C_VEL
LIN {X 0,Y 510.252,Z 268.436,A -85,B 0,C 180,E1 -5505.604,E2 -5505.604} C_VEL
LIN {X 0,Y 510.76,Z 247.14,A -85,B 0,C 180,E1 -5508.864,E2 -5508.864} C_VEL
LIN {X 0,Y 511.293,Z 228.327,A -85,B 0,C 180,E1 -5511.783,E2 -5511.783} C_VEL
LIN {X 0,Y 511.723,Z 216.237,A -85,B 0,C 180,E1 -5513.683,E2 -5513.683} C_VEL
LIN {X 0,Y 509.922,Z 205.969,A -85,B 0,C 180,E1 -5515.454,E2 -5515.454} C_VEL
LIN {X 0,Y 509.883,Z 205.976,A -85,B 0,C 180,E1 -5518.097,E2 -5518.097} C_VEL
LIN {X 0,Y 509.832,Z 205.975,A -85,B 0,C 180,E1 -5521.277,E2 -5521.277} C_VEL
LIN {X 0,Y 509.843,Z 205.978,A -85,B 0,C 180,E1 -5524.2,E2 -5524.2} C_VEL
LIN {X 0,Y 509.8,Z 205.979,A -85,B 0,C 180,E1 -5527.337,E2 -5527.337} C_VEL
LIN {X 0,Y 509.816,Z 205.977,A -85,B 0,C 180,E1 -5530.379,E2 -5530.379} C_VEL
LIN {X 0,Y 509.798,Z 205.978,A -85,B 0,C 180,E1 -5533.059,E2 -5533.059} C_VEL
LIN {X 0,Y 509.804,Z 205.986,A -85,B 0,C 180,E1 -5535.789,E2 -5535.789} C_VEL
LIN {X 0,Y 509.828,Z 205.974,A -85,B 0,C 180,E1 -5538.571,E2 -5538.571} C_VEL
LIN {X 0,Y 509.817,Z 205.982,A -85,B 0,C 180,E1 -5541.783,E2 -5541.783} C_VEL
LIN {X 0,Y 509.809,Z 205.976,A -85,B 0,C 180,E1 -5544.62,E2 -5544.62} C_VEL
LIN {X 0,Y 509.827,Z 205.982,A -85,B 0,C 180,E1 -5547.478,E2 -5547.478} C_VEL
LIN {X 0,Y 509.817,Z 205.975,A -85,B 0,C 180,E1 -5550.271,E2 -5550.271} C_VEL
LIN {X 0,Y 509.843,Z 205.974,A -85,B 0,C 180,E1 -5552.942,E2 -5552.942} C_VEL
LIN {X 0,Y 509.828,Z 205.98,A -85,B 0,C 180,E1 -5555.572,E2 -5555.572} C_VEL
LIN {X 0,Y 509.8,Z 205.977,A -85,B 0,C 180,E1 -5558.147,E2 -5558.147} C_VEL
LIN {X 0,Y 509.817,Z 205.976,A -85,B 0,C 180,E1 -5560.679,E2 -5560.679} C_VEL
LIN {X 0,Y 509.85,Z 205.979,A -85,B 0,C 180,E1 -5563.173,E2 -5563.173} C_VEL
LIN {X 0,Y 509.81,Z 205.979,A -85,B 0,C 180,E1 -5565.632,E2 -5565.632} C_VEL
LIN {X 0,Y 509.88,Z 205.972,A -85,B 0,C 180,E1 -5568.874,E2 -5568.874} C_VEL
LIN {X 0,Y 509.897,Z 205.965,A -85,B 0,C 180,E1 -5572.077,E2 -5572.077} C_VEL
LIN {X 0,Y 509.925,Z 205.963,A -85,B 0,C 180,E1 -5574.463,E2 -5574.463} C_VEL
LIN {X 0,Y 509.997,Z 205.954,A -85,B 0,C 180,E1 -5577.63,E2 -5577.63} C_VEL
LIN {X 0,Y 509.994,Z 205.953,A -85,B 0,C 180,E1 -5580,E2 -5580} C_VEL
LIN {X 0,Y 509.998,Z 205.954,A -85,B 0,C 180,E1 -5582.369,E2 -5582.369} C_VEL
LIN {X 0,Y 509.957,Z 205.958,A -85,B 0,C 180,E1 -5585.536,E2 -5585.536} C_VEL
LIN {X 0,Y 509.903,Z 205.964,A -85,B 0,C 180,E1 -5587.922,E2 -5587.922} C_VEL
LIN {X 0,Y 509.881,Z 205.97,A -85,B 0,C 180,E1 -5591.126,E2 -5591.126} C_VEL
LIN {X 0,Y 509.825,Z 205.974,A -85,B 0,C 180,E1 -5593.553,E2 -5593.553} C_VEL
LIN {X 0,Y 509.813,Z 205.977,A -85,B 0,C 180,E1 -5596.004,E2 -5596.004} C_VEL
LIN {X 0,Y 509.82,Z 205.982,A -85,B 0,C 180,E1 -5598.485,E2 -5598.485} C_VEL
LIN {X 0,Y 509.828,Z 205.976,A -85,B 0,C 180,E1 -5601.002,E2 -5601.002} C_VEL
LIN {X 0,Y 509.823,Z 205.974,A -85,B 0,C 180,E1 -5603.563,E2 -5603.563} C_VEL
LIN {X 0,Y 509.867,Z 205.977,A -85,B 0,C 180,E1 -5606.381,E2 -5606.381} C_VEL
LIN {X 0,Y 509.846,Z 205.974,A -85,B 0,C 180,E1 -5608.846,E2 -5608.846} C_VEL
LIN {X 0,Y 509.784,Z 205.98,A -85,B 0,C 180,E1 -5611.592,E2 -5611.592} C_VEL
LIN {X 0,Y 509.814,Z 205.982,A -85,B 0,C 180,E1 -5614.416,E2 -5614.416} C_VEL
LIN {X 0,Y 509.783,Z 205.979,A -85,B 0,C 180,E1 -5617.343,E2 -5617.343} C_VEL
LIN {X 0,Y 509.847,Z 205.977,A -85,B 0,C 180,E1 -5620.381,E2 -5620.381} C_VEL
LIN {X 0,Y 509.808,Z 205.976,A -85,B 0,C 180,E1 -5623.067,E2 -5623.067} C_VEL
LIN {X 0,Y 509.801,Z 205.982,A -85,B 0,C 180,E1 -5625.795,E2 -5625.795} C_VEL
LIN {X 0,Y 509.84,Z 205.974,A -85,B 0,C 180,E1 -5628.579,E2 -5628.579} C_VEL
LIN {X 0,Y 509.829,Z 205.98,A -85,B 0,C 180,E1 -5631.789,E2 -5631.789} C_VEL
LIN {X 0,Y 509.808,Z 205.98,A -85,B 0,C 180,E1 -5633.784,E2 -5633.784} C_VEL
LIN {X 0,Y 509.145,Z 206.061,A -85,B 0,C 180,E1 -5634.444,E2 -5634.444} C_VEL
LIN {X 0,Y 506.326,Z 206.414,A -85,B 0,C 180,E1 -5635.516,E2 -5635.516} C_VEL
LIN {X 0,Y 503.931,Z 206.71,A -85,B 0,C 180,E1 -5636.379,E2 -5636.379} C_VEL
LIN {X 0,Y 502.884,Z 206.839,A -85,B 0,C 180,E1 -5637.046,E2 -5637.046} C_VEL
LIN {X 0,Y 502.788,Z 206.851,A -85,B 0,C 180,E1 -5637.271,E2 -5637.271} C_VEL
LIN {X 0,Y 502.815,Z 206.852,A -85,B 0,C 180,E1 -5640.065,E2 -5640.065} C_VEL
LIN {X 0,Y 502.822,Z 206.847,A -85,B 0,C 180,E1 -5642.536,E2 -5642.536} C_VEL
LIN {X 0,Y 502.818,Z 206.85,A -85,B 0,C 180,E1 -5645.301,E2 -5645.301} C_VEL
LIN {X 0,Y 502.775,Z 206.858,A -85,B 0,C 180,E1 -5647.829,E2 -5647.829} C_VEL
LIN {X 0,Y 502.817,Z 206.847,A -85,B 0,C 180,E1 -5650.402,E2 -5650.402} C_VEL
LIN {X 0,Y 502.828,Z 206.847,A -85,B 0,C 180,E1 -5652.933,E2 -5652.933} C_VEL
LIN {X 0,Y 502.847,Z 206.851,A -85,B 0,C 180,E1 -5655.431,E2 -5655.431} C_VEL
LIN {X 0,Y 502.874,Z 206.841,A -85,B 0,C 180,E1 -5658.718,E2 -5658.718} C_VEL
LIN {X 0,Y 502.9,Z 206.838,A -85,B 0,C 180,E1 -5661.968,E2 -5661.968} C_VEL
LIN {X 0,Y 502.932,Z 206.833,A -85,B 0,C 180,E1 -5664.387,E2 -5664.387} C_VEL
LIN {X 0,Y 503.024,Z 206.825,A -85,B 0,C 180,E1 -5667.598,E2 -5667.598} C_VEL
LIN {X 0,Y 503.027,Z 206.821,A -85,B 0,C 180,E1 -5670,E2 -5670} C_VEL
LIN {X 0,Y 503.024,Z 206.822,A -85,B 0,C 180,E1 -5672.402,E2 -5672.402} C_VEL
LIN {X 0,Y 502.93,Z 206.835,A -85,B 0,C 180,E1 -5675.613,E2 -5675.613} C_VEL
LIN {X 0,Y 502.9,Z 206.837,A -85,B 0,C 180,E1 -5678.033,E2 -5678.033} C_VEL
LIN {X 0,Y 502.874,Z 206.844,A -85,B 0,C 180,E1 -5681.282,E2 -5681.282} C_VEL
LIN {X 0,Y 502.84,Z 206.848,A -85,B 0,C 180,E1 -5684.569,E2 -5684.569} C_VEL
LIN {X 0,Y 502.856,Z 206.842,A -85,B 0,C 180,E1 -5687.905,E2 -5687.905} C_VEL
LIN {X 0,Y 502.821,Z 206.851,A -85,B 0,C 180,E1 -5690.534,E2 -5690.534} C_VEL
LIN {X 0,Y 502.788,Z 206.855,A -85,B 0,C 180,E1 -5693.038,E2 -5693.038} C_VEL
LIN {X 0,Y 502.831,Z 206.847,A -85,B 0,C 180,E1 -5695.673,E2 -5695.673} C_VEL
LIN {X 0,Y 502.829,Z 206.852,A -85,B 0,C 180,E1 -5698.37,E2 -5698.37} C_VEL
LIN {X 0,Y 502.91,Z 206.916,A -85,B 0,C 180,E1 -5700.694,E2 -5700.694} C_VEL
LIN {X 0,Y 503.486,Z 212.187,A -85,B 0,C 180,E1 -5701.781,E2 -5701.781} C_VEL
LIN {X 0,Y 503.263,Z 224.598,A -85,B 0,C 180,E1 -5704.253,E2 -5704.253} C_VEL
LIN {X 0,Y 505.42,Z 236.304,A -85,B 0,C 180,E1 -5704.51,E2 -5704.51} C_VEL
LIN {X 0,Y 504.773,Z 331.978,A -85,B 0,C 180,E1 -5705.929,E2 -5705.929} C_VEL
LIN {X 0,Y 504.553,Z 345.05,A -85,B 0,C 180,E1 -5706.285,E2 -5706.285} C_VEL
LIN {X 0,Y 504.363,Z 357.899,A -85,B 0,C 180,E1 -5706.806,E2 -5706.806} C_VEL
LIN {X 0,Y 504.015,Z 370.052,A -85,B 0,C 180,E1 -5707.48,E2 -5707.48} C_VEL
LIN {X 0,Y 503.694,Z 380.87,A -85,B 0,C 180,E1 -5708.248,E2 -5708.248} C_VEL
LIN {X 0,Y 503.346,Z 391.4,A -85,B 0,C 180,E1 -5709.178,E2 -5709.178} C_VEL
LIN {X 0,Y 503.027,Z 400.987,A -85,B 0,C 180,E1 -5710.235,E2 -5710.235} C_VEL
LIN {X 0,Y 502.765,Z 409.093,A -85,B 0,C 180,E1 -5711.332,E2 -5711.332} C_VEL
LIN {X 0,Y 502.495,Z 415.783,A -85,B 0,C 180,E1 -5712.435,E2 -5712.435} C_VEL
LIN {X 0,Y 502.356,Z 422.509,A -85,B 0,C 180,E1 -5713.827,E2 -5713.827} C_VEL
LIN {X 0,Y 502.255,Z 427.02,A -85,B 0,C 180,E1 -5715.036,E2 -5715.036} C_VEL
LIN {X 0,Y 502.156,Z 430.216,A -85,B 0,C 180,E1 -5716.15,E2 -5716.15} C_VEL
LIN {X 0,Y 502.07,Z 433.365,A -85,B 0,C 180,E1 -5717.786,E2 -5717.786} C_VEL
LIN {X 0,Y 502.035,Z 434.676,A -85,B 0,C 180,E1 -5719.101,E2 -5719.101} C_VEL
LIN {X 0,Y 502.019,Z 434.933,A -85,B 0,C 180,E1 -5720.344,E2 -5720.344} C_VEL
LIN {X 0,Y 502.011,Z 433.853,A -85,B 0,C 180,E1 -5721.977,E2 -5721.977} C_VEL
LIN {X 0,Y 502.126,Z 431.288,A -85,B 0,C 180,E1 -5723.498,E2 -5723.498} C_VEL
LIN {X 0,Y 502.181,Z 427.332,A -85,B 0,C 180,E1 -5724.985,E2 -5724.985} C_VEL
LIN {X 0,Y 502.305,Z 422.846,A -85,B 0,C 180,E1 -5726.21,E2 -5726.21} C_VEL
LIN {X 0,Y 502.507,Z 416.897,A -85,B 0,C 180,E1 -5727.476,E2 -5727.476} C_VEL
LIN {X 0,Y 502.762,Z 409.744,A -85,B 0,C 180,E1 -5728.683,E2 -5728.683} C_VEL
LIN {X 0,Y 503.012,Z 401.577,A -85,B 0,C 180,E1 -5729.803,E2 -5729.803} C_VEL
LIN {X 0,Y 503.367,Z 392.136,A -85,B 0,C 180,E1 -5730.856,E2 -5730.856} C_VEL
LIN {X 0,Y 503.638,Z 381.735,A -85,B 0,C 180,E1 -5731.79,E2 -5731.79} C_VEL
LIN {X 0,Y 504.004,Z 370.366,A -85,B 0,C 180,E1 -5732.603,E2 -5732.603} C_VEL
LIN {X 0,Y 504.317,Z 358.944,A -85,B 0,C 180,E1 -5733.243,E2 -5733.243} C_VEL
LIN {X 0,Y 504.604,Z 346.235,A -85,B 0,C 180,E1 -5733.77,E2 -5733.77} C_VEL
LIN {X 0,Y 504.774,Z 332.435,A -85,B 0,C 180,E1 -5734.154,E2 -5734.154} C_VEL
LIN {X 0,Y 505.457,Z 235.949,A -85,B 0,C 180,E1 -5735.593,E2 -5735.593} C_VEL
LIN {X 0,Y 503.284,Z 224.586,A -85,B 0,C 180,E1 -5735.838,E2 -5735.838} C_VEL
LIN {X 0,Y 503.256,Z 209.737,A -85,B 0,C 180,E1 -5738.495,E2 -5738.495} C_VEL
LIN {X 0,Y 502.861,Z 206.85,A -85,B 0,C 180,E1 -5739.065,E2 -5739.065} C_VEL
LIN {X 0,Y 502.829,Z 206.849,A -85,B 0,C 180,E1 -5742.092,E2 -5742.092} C_VEL
LIN {X 0,Y 502.801,Z 206.859,A -85,B 0,C 180,E1 -5745.428,E2 -5745.428} C_VEL
LIN {X 0,Y 502.85,Z 206.849,A -85,B 0,C 180,E1 -5748.716,E2 -5748.716} C_VEL
LIN {X 0,Y 502.853,Z 206.845,A -85,B 0,C 180,E1 -5751.966,E2 -5751.966} C_VEL
LIN {X 0,Y 502.911,Z 206.837,A -85,B 0,C 180,E1 -5754.386,E2 -5754.386} C_VEL
LIN {X 0,Y 502.97,Z 206.832,A -85,B 0,C 180,E1 -5757.598,E2 -5757.598} C_VEL
LIN {X 0,Y 502.967,Z 206.83,A -85,B 0,C 180,E1 -5760,E2 -5760} C_VEL
LIN {X 0,Y 502.968,Z 206.831,A -85,B 0,C 180,E1 -5762.403,E2 -5762.403} C_VEL
LIN {X 0,Y 502.879,Z 206.84,A -85,B 0,C 180,E1 -5765.614,E2 -5765.614} C_VEL
LIN {X 0,Y 502.849,Z 206.844,A -85,B 0,C 180,E1 -5768.034,E2 -5768.034} C_VEL
LIN {X 0,Y 502.849,Z 206.846,A -85,B 0,C 180,E1 -5771.284,E2 -5771.284} C_VEL
LIN {X 0,Y 502.793,Z 206.855,A -85,B 0,C 180,E1 -5774.573,E2 -5774.573} C_VEL
LIN {X 0,Y 502.814,Z 206.847,A -85,B 0,C 180,E1 -5777.909,E2 -5777.909} C_VEL
LIN {X 0,Y 502.782,Z 206.857,A -85,B 0,C 180,E1 -5780.538,E2 -5780.538} C_VEL
LIN {X 0,Y 502.76,Z 206.855,A -85,B 0,C 180,E1 -5783.042,E2 -5783.042} C_VEL
LIN {X 0,Y 502.797,Z 206.85,A -85,B 0,C 180,E1 -5785.678,E2 -5785.678} C_VEL
LIN {X 0,Y 502.8,Z 206.856,A -85,B 0,C 180,E1 -5788.375,E2 -5788.375} C_VEL
LIN {X 0,Y 502.757,Z 206.855,A -85,B 0,C 180,E1 -5791.502,E2 -5791.502} C_VEL
LIN {X 0,Y 502.769,Z 206.86,A -85,B 0,C 180,E1 -5794.447,E2 -5794.447} C_VEL
LIN {X 0,Y 502.747,Z 206.857,A -85,B 0,C 180,E1 -5797.181,E2 -5797.181} C_VEL
LIN {X 0,Y 502.757,Z 206.86,A -85,B 0,C 180,E1 -5800.019,E2 -5800.019} C_VEL
LIN {X 0,Y 502.775,Z 206.861,A -85,B 0,C 180,E1 -5802.203,E2 -5802.203} C_VEL
LIN {X 0,Y 502.76,Z 206.855,A -85,B 0,C 180,E1 -5805.473,E2 -5805.473} C_VEL
LIN {X 0,Y 502.799,Z 206.85,A -85,B 0,C 180,E1 -5808.937,E2 -5808.937} C_VEL
LIN {X 0,Y 502.774,Z 206.86,A -85,B 0,C 180,E1 -5812.049,E2 -5812.049} C_VEL
LIN {X 0,Y 502.792,Z 206.851,A -85,B 0,C 180,E1 -5815.038,E2 -5815.038} C_VEL
LIN {X 0,Y 502.77,Z 206.861,A -85,B 0,C 180,E1 -5817.918,E2 -5817.918} C_VEL
LIN {X 0,Y 502.813,Z 206.852,A -85,B 0,C 180,E1 -5820.715,E2 -5820.715} C_VEL
LIN {X 0,Y 502.855,Z 206.85,A -85,B 0,C 180,E1 -5823.442,E2 -5823.442} C_VEL
LIN {X 0,Y 502.851,Z 206.851,A -85,B 0,C 180,E1 -5824.772,E2 -5824.772} C_VEL
LIN {X 0,Y 504.434,Z 216.654,A -85,B 0,C 180,E1 -5826.38,E2 -5826.38} C_VEL
LIN {X 0,Y 503.947,Z 235.936,A -85,B 0,C 180,E1 -5829.359,E2 -5829.359} C_VEL
LIN {X 0,Y 503.445,Z 256.755,A -85,B 0,C 180,E1 -5832.536,E2 -5832.536} C_VEL
LIN {X 0,Y 503.184,Z 267.615,A -85,B 0,C 180,E1 -5834.182,E2 -5834.182} C_VEL
LIN {X 0,Y 505.29,Z 283.197,A -85,B 0,C 180,E1 -5834.489,E2 -5834.489} C_VEL
LIN {X 0,Y 504.73,Z 376.578,A -85,B 0,C 180,E1 -5835.872,E2 -5835.872} C_VEL
LIN {X 0,Y 504.445,Z 389.787,A -85,B 0,C 180,E1 -5836.224,E2 -5836.224} C_VEL
LIN {X 0,Y 504.122,Z 401.958,A -85,B 0,C 180,E1 -5836.703,E2 -5836.703} C_VEL
LIN {X 0,Y 503.776,Z 414.371,A -85,B 0,C 180,E1 -5837.366,E2 -5837.366} C_VEL
LIN {X 0,Y 503.434,Z 425.274,A -85,B 0,C 180,E1 -5838.118,E2 -5838.118} C_VEL
LIN {X 0,Y 503.075,Z 435.889,A -85,B 0,C 180,E1 -5839.028,E2 -5839.028} C_VEL
LIN {X 0,Y 502.811,Z 444.572,A -85,B 0,C 180,E1 -5839.939,E2 -5839.939} C_VEL
LIN {X 0,Y 502.606,Z 452.58,A -85,B 0,C 180,E1 -5840.95,E2 -5840.95} C_VEL
LIN {X 0,Y 502.368,Z 460.403,A -85,B 0,C 180,E1 -5842.161,E2 -5842.161} C_VEL
LIN {X 0,Y 502.235,Z 467.602,A -85,B 0,C 180,E1 -5843.573,E2 -5843.573} C_VEL
LIN {X 0,Y 502.171,Z 472.397,A -85,B 0,C 180,E1 -5844.781,E2 -5844.781} C_VEL
LIN {X 0,Y 502.164,Z 476.064,A -85,B 0,C 180,E1 -5845.988,E2 -5845.988} C_VEL
LIN {X 0,Y 502.123,Z 477.956,A -85,B 0,C 180,E1 -5846.791,E2 -5846.791} C_VEL
LIN {X 0,Y 502.121,Z 479.375,A -85,B 0,C 180,E1 -5847.594,E2 -5847.594} C_VEL
LIN {X 0,Y 501.997,Z 481.009,A -85,B 0,C 180,E1 -5849.198,E2 -5849.198} C_VEL
LIN {X 0,Y 501.992,Z 481.235,A -85,B 0,C 180,E1 -5850,E2 -5850} C_VEL
LIN {X 0,Y 502.036,Z 480.417,A -85,B 0,C 180,E1 -5851.604,E2 -5851.604} C_VEL
LIN {X 0,Y 502.121,Z 479.421,A -85,B 0,C 180,E1 -5852.406,E2 -5852.406} C_VEL
LIN {X 0,Y 502.12,Z 478.014,A -85,B 0,C 180,E1 -5853.209,E2 -5853.209} C_VEL
LIN {X 0,Y 502.102,Z 475.054,A -85,B 0,C 180,E1 -5854.415,E2 -5854.415} C_VEL
LIN {X 0,Y 502.199,Z 471.047,A -85,B 0,C 180,E1 -5855.621,E2 -5855.621} C_VEL
LIN {X 0,Y 502.289,Z 464.975,A -85,B 0,C 180,E1 -5857.011,E2 -5857.011} C_VEL
LIN {X 0,Y 502.46,Z 458.131,A -85,B 0,C 180,E1 -5858.242,E2 -5858.242} C_VEL
LIN {X 0,Y 502.669,Z 449.766,A -85,B 0,C 180,E1 -5859.454,E2 -5859.454} C_VEL
LIN {X 0,Y 502.941,Z 441.166,A -85,B 0,C 180,E1 -5860.465,E2 -5860.465} C_VEL
LIN {X 0,Y 503.337,Z 430.557,A -85,B 0,C 180,E1 -5861.475,E2 -5861.475} C_VEL
LIN {X 0,Y 503.677,Z 419.251,A -85,B 0,C 180,E1 -5862.341,E2 -5862.341} C_VEL
LIN {X 0,Y 503.972,Z 408.477,A -85,B 0,C 180,E1 -5862.993,E2 -5862.993} C_VEL
LIN {X 0,Y 504.265,Z 396.48,A -85,B 0,C 180,E1 -5863.55,E2 -5863.55} C_VEL
LIN {X 0,Y 504.612,Z 383.544,A -85,B 0,C 180,E1 -5863.977,E2 -5863.977} C_VEL
LIN {X 0,Y 504.838,Z 369.848,A -85,B 0,C 180,E1 -5864.253,E2 -5864.253} C_VEL
LIN {X 0,Y 505.179,Z 281.372,A -85,B 0,C 180,E1 -5865.549,E2 -5865.549} C_VEL
LIN {X 0,Y 503.231,Z 268.166,A -85,B 0,C 180,E1 -5865.822,E2 -5865.822} C_VEL
LIN {X 0,Y 503.775,Z 248.182,A -85,B 0,C 180,E1 -5868.924,E2 -5868.924} C_VEL
LIN {X 0,Y 504.338,Z 229.39,A -85,B 0,C 180,E1 -5871.884,E2 -5871.884} C_VEL
LIN {X 0,Y 504.789,Z 217.289,A -85,B 0,C 180,E1 -5873.81,E2 -5873.81} C_VEL
LIN {X 0,Y 502.882,Z 206.847,A -85,B 0,C 180,E1 -5875.617,E2 -5875.617} C_VEL
LIN {X 0,Y 502.828,Z 206.853,A -85,B 0,C 180,E1 -5878.37,E2 -5878.37} C_VEL
LIN {X 0,Y 502.779,Z 206.855,A -85,B 0,C 180,E1 -5881.496,E2 -5881.496} C_VEL
LIN {X 0,Y 502.791,Z 206.859,A -85,B 0,C 180,E1 -5883.99,E2 -5883.99} C_VEL
LIN {X 0,Y 502.762,Z 206.854,A -85,B 0,C 180,E1 -5887.175,E2 -5887.175} C_VEL
LIN {X 0,Y 502.766,Z 206.86,A -85,B 0,C 180,E1 -5890.012,E2 -5890.012} C_VEL
LIN {X 0,Y 502.779,Z 206.855,A -85,B 0,C 180,E1 -5892.196,E2 -5892.196} C_VEL
LIN {X 0,Y 502.774,Z 206.857,A -85,B 0,C 180,E1 -5895.465,E2 -5895.465} C_VEL
LIN {X 0,Y 502.79,Z 206.851,A -85,B 0,C 180,E1 -5898.931,E2 -5898.931} C_VEL
LIN {X 0,Y 502.759,Z 206.858,A -85,B 0,C 180,E1 -5902.043,E2 -5902.043} C_VEL
LIN {X 0,Y 502.773,Z 206.854,A -85,B 0,C 180,E1 -5905.032,E2 -5905.032} C_VEL
LIN {X 0,Y 502.748,Z 206.859,A -85,B 0,C 180,E1 -5907.913,E2 -5907.913} C_VEL
LIN {X 0,Y 502.783,Z 206.852,A -85,B 0,C 180,E1 -5910.709,E2 -5910.709} C_VEL
LIN {X 0,Y 502.819,Z 206.856,A -85,B 0,C 180,E1 -5913.436,E2 -5913.436} C_VEL
LIN {X 0,Y 502.754,Z 206.856,A -85,B 0,C 180,E1 -5916.084,E2 -5916.084} C_VEL
LIN {X 0,Y 502.748,Z 206.857,A -85,B 0,C 180,E1 -5918.687,E2 -5918.687} C_VEL
LIN {X 0,Y 502.796,Z 206.851,A -85,B 0,C 180,E1 -5921.876,E2 -5921.876} C_VEL
LIN {X 0,Y 502.789,Z 206.852,A -85,B 0,C 180,E1 -5924.661,E2 -5924.661} C_VEL
LIN {X 0,Y 502.847,Z 206.843,A -85,B 0,C 180,E1 -5928.025,E2 -5928.025} C_VEL
LIN {X 0,Y 502.824,Z 206.854,A -85,B 0,C 180,E1 -5931.156,E2 -5931.156} C_VEL
LIN {X 0,Y 502.85,Z 206.845,A -85,B 0,C 180,E1 -5933.58,E2 -5933.58} C_VEL
LIN {X 0,Y 502.849,Z 206.849,A -85,B 0,C 180,E1 -5936.795,E2 -5936.795} C_VEL
LIN {X 0,Y 502.982,Z 206.832,A -85,B 0,C 180,E1 -5939.199,E2 -5939.199} C_VEL
LIN {X 0,Y 502.848,Z 206.844,A -85,B 0,C 180,E1 -5941.601,E2 -5941.601} C_VEL
LIN {X 0,Y 502.851,Z 206.847,A -85,B 0,C 180,E1 -5943.205,E2 -5943.205} C_VEL
LIN {X 0,Y 502.892,Z 206.841,A -85,B 0,C 180,E1 -5946.419,E2 -5946.419} C_VEL
LIN {X 0,Y 502.825,Z 206.854,A -85,B 0,C 180,E1 -5948.844,E2 -5948.844} C_VEL
LIN {X 0,Y 502.843,Z 206.845,A -85,B 0,C 180,E1 -5952.101,E2 -5952.101} C_VEL
LIN {X 0,Y 502.797,Z 206.85,A -85,B 0,C 180,E1 -5955.401,E2 -5955.401} C_VEL
LIN {X 0,Y 502.796,Z 206.852,A -85,B 0,C 180,E1 -5958.124,E2 -5958.124} C_VEL
LIN {X 0,Y 502.773,Z 206.853,A -85,B 0,C 180,E1 -5961.311,E2 -5961.311} C_VEL
LIN {X 0,Y 502.774,Z 206.854,A -85,B 0,C 180,E1 -5963.914,E2 -5963.914} C_VEL
LIN {X 0,Y 502.836,Z 206.851,A -85,B 0,C 180,E1 -5966.567,E2 -5966.567} C_VEL
LIN {X 0,Y 502.798,Z 206.849,A -85,B 0,C 180,E1 -5969.289,E2 -5969.289} C_VEL
LIN {X 0,Y 502.746,Z 206.861,A -85,B 0,C 180,E1 -5972.087,E2 -5972.087} C_VEL
LIN {X 0,Y 502.771,Z 206.853,A -85,B 0,C 180,E1 -5974.968,E2 -5974.968} C_VEL
LIN {X 0,Y 502.761,Z 206.859,A -85,B 0,C 180,E1 -5977.956,E2 -5977.956} C_VEL
LIN {X 0,Y 502.799,Z 206.849,A -85,B 0,C 180,E1 -5981,E2 -5981} C_VEL
LIN {X 0,Y 502.75,Z 206.856,A -85,B 0,C 180,E1 -5983.379,E2 -5983.379} C_VEL
LIN {X 0,Y 502.76,Z 206.857,A -85,B 0,C 180,E1 -5985.664,E2 -5985.664} C_VEL
LIN {X 0,Y 502.804,Z 206.849,A -85,B 0,C 180,E1 -5989.007,E2 -5989.007} C_VEL
LIN {X 0,Y 502.771,Z 206.86,A -85,B 0,C 180,E1 -5992.049,E2 -5992.049} C_VEL
LIN {X 0,Y 502.79,Z 206.851,A -85,B 0,C 180,E1 -5995.038,E2 -5995.038} C_VEL
LIN {X 0,Y 502.788,Z 206.851,A -85,B 0,C 180,E1 -5997.271,E2 -5997.271} C_VEL
LIN {X 0,Y 502.093,Z 206.944,A -85,B 0,C 180,E1 -5997.94,E2 -5997.94} C_VEL
LIN {X 0,Y 499.235,Z 207.296,A -85,B 0,C 180,E1 -5999.026,E2 -5999.026} C_VEL
LIN {X 0,Y 496.843,Z 207.598,A -85,B 0,C 180,E1 -5999.901,E2 -5999.901} C_VEL
LIN {X 0,Y 495.827,Z 207.719,A -85,B 0,C 180,E1 -6000.577,E2 -6000.577} C_VEL
LIN {X 0,Y 495.749,Z 207.727,A -85,B 0,C 180,E1 -6000.805,E2 -6000.805} C_VEL
LIN {X 0,Y 495.788,Z 207.728,A -85,B 0,C 180,E1 -6003.935,E2 -6003.935} C_VEL
LIN {X 0,Y 495.756,Z 207.729,A -85,B 0,C 180,E1 -6007.14,E2 -6007.14} C_VEL
LIN {X 0,Y 495.763,Z 207.728,A -85,B 0,C 180,E1 -6010.112,E2 -6010.112} C_VEL
LIN {X 0,Y 495.78,Z 207.724,A -85,B 0,C 180,E1 -6012.683,E2 -6012.683} C_VEL
LIN {X 0,Y 495.789,Z 207.727,A -85,B 0,C 180,E1 -6015.219,E2 -6015.219} C_VEL
LIN {X 0,Y 495.848,Z 207.715,A -85,B 0,C 180,E1 -6018.556,E2 -6018.556} C_VEL
LIN {X 0,Y 495.871,Z 207.715,A -85,B 0,C 180,E1 -6021.853,E2 -6021.853} C_VEL
LIN {X 0,Y 495.888,Z 207.71,A -85,B 0,C 180,E1 -6024.307,E2 -6024.307} C_VEL
LIN {X 0,Y 495.993,Z 207.701,A -85,B 0,C 180,E1 -6027.564,E2 -6027.564} C_VEL
LIN {X 0,Y 495.998,Z 207.697,A -85,B 0,C 180,E1 -6030,E2 -6030} C_VEL
LIN {X 0,Y 495.993,Z 207.698,A -85,B 0,C 180,E1 -6032.436,E2 -6032.436} C_VEL
LIN {X 0,Y 495.885,Z 207.712,A -85,B 0,C 180,E1 -6035.693,E2 -6035.693} C_VEL
LIN {X 0,Y 495.871,Z 207.712,A -85,B 0,C 180,E1 -6038.147,E2 -6038.147} C_VEL
LIN {X 0,Y 495.849,Z 207.718,A -85,B 0,C 180,E1 -6041.444,E2 -6041.444} C_VEL
LIN {X 0,Y 495.785,Z 207.73,A -85,B 0,C 180,E1 -6044.781,E2 -6044.781} C_VEL
LIN {X 0,Y 495.781,Z 207.726,A -85,B 0,C 180,E1 -6047.317,E2 -6047.317} C_VEL
LIN {X 0,Y 495.771,Z 207.725,A -85,B 0,C 180,E1 -6049.888,E2 -6049.888} C_VEL
LIN {X 0,Y 495.749,Z 207.735,A -85,B 0,C 180,E1 -6052.858,E2 -6052.858} C_VEL
LIN {X 0,Y 495.788,Z 207.726,A -85,B 0,C 180,E1 -6056.065,E2 -6056.065} C_VEL
LIN {X 0,Y 495.769,Z 207.733,A -85,B 0,C 180,E1 -6058.812,E2 -6058.812} C_VEL
LIN {X 0,Y 495.85,Z 207.778,A -85,B 0,C 180,E1 -6060.553,E2 -6060.553} C_VEL
LIN {X 0,Y 496.49,Z 212.693,A -85,B 0,C 180,E1 -6061.58,E2 -6061.58} C_VEL
LIN {X 0,Y 496.267,Z 224.948,A -85,B 0,C 180,E1 -6064.04,E2 -6064.04} C_VEL
LIN {X 0,Y 498.523,Z 236.551,A -85,B 0,C 180,E1 -6064.292,E2 -6064.292} C_VEL
LIN {X 0,Y 497.89,Z 331.972,A -85,B 0,C 180,E1 -6065.73,E2 -6065.73} C_VEL
LIN {X 0,Y 497.678,Z 345.117,A -85,B 0,C 180,E1 -6066.091,E2 -6066.091} C_VEL
LIN {X 0,Y 497.474,Z 357.158,A -85,B 0,C 180,E1 -6066.579,E2 -6066.579} C_VEL
LIN {X 0,Y 497.115,Z 369.322,A -85,B 0,C 180,E1 -6067.243,E2 -6067.243} C_VEL
LIN {X 0,Y 496.738,Z 380.449,A -85,B 0,C 180,E1 -6068.03,E2 -6068.03} C_VEL
LIN {X 0,Y 496.38,Z 391.34,A -85,B 0,C 180,E1 -6068.995,E2 -6068.995} C_VEL
LIN {X 0,Y 496.039,Z 401.165,A -85,B 0,C 180,E1 -6070.086,E2 -6070.086} C_VEL
LIN {X 0,Y 495.724,Z 409.903,A -85,B 0,C 180,E1 -6071.289,E2 -6071.289} C_VEL
LIN {X 0,Y 495.426,Z 417.817,A -85,B 0,C 180,E1 -6072.658,E2 -6072.658} C_VEL
LIN {X 0,Y 495.266,Z 424.031,A -85,B 0,C 180,E1 -6074.047,E2 -6074.047} C_VEL
LIN {X 0,Y 495.129,Z 429.149,A -85,B 0,C 180,E1 -6075.568,E2 -6075.568} C_VEL
LIN {X 0,Y 495.023,Z 432.537,A -85,B 0,C 180,E1 -6077.042,E2 -6077.042} C_VEL
LIN {X 0,Y 494.975,Z 434.196,A -85,B 0,C 180,E1 -6078.138,E2 -6078.138} C_VEL
LIN {X 0,Y 494.938,Z 435.078,A -85,B 0,C 180,E1 -6079.218,E2 -6079.218} C_VEL
LIN {X 0,Y 494.927,Z 435.272,A -85,B 0,C 180,E1 -6080.283,E2 -6080.283} C_VEL
LIN {X 0,Y 494.938,Z 434.82,A -85,B 0,C 180,E1 -6081.343,E2 -6081.343} C_VEL
LIN {X 0,Y 494.947,Z 433.279,A -85,B 0,C 180,E1 -6082.663,E2 -6082.663} C_VEL
LIN {X 0,Y 495.096,Z 430.594,A -85,B 0,C 180,E1 -6084.002,E2 -6084.002} C_VEL
LIN {X 0,Y 495.124,Z 426.499,A -85,B 0,C 180,E1 -6085.405,E2 -6085.405} C_VEL
LIN {X 0,Y 495.358,Z 420.89,A -85,B 0,C 180,E1 -6086.823,E2 -6086.823} C_VEL
LIN {X 0,Y 495.566,Z 414.319,A -85,B 0,C 180,E1 -6088.112,E2 -6088.112} C_VEL
LIN {X 0,Y 495.861,Z 406.559,A -85,B 0,C 180,E1 -6089.321,E2 -6089.321} C_VEL
LIN {X 0,Y 496.242,Z 397.012,A -85,B 0,C 180,E1 -6090.519,E2 -6090.519} C_VEL
LIN {X 0,Y 496.538,Z 386.576,A -85,B 0,C 180,E1 -6091.566,E2 -6091.566} C_VEL
LIN {X 0,Y 496.921,Z 375.002,A -85,B 0,C 180,E1 -6092.488,E2 -6092.488} C_VEL
LIN {X 0,Y 497.395,Z 362.941,A -85,B 0,C 180,E1 -6093.232,E2 -6093.232} C_VEL
LIN {X 0,Y 497.618,Z 351.94,A -85,B 0,C 180,E1 -6093.754,E2 -6093.754} C_VEL
LIN {X 0,Y 497.831,Z 338.271,A -85,B 0,C 180,E1 -6094.217,E2 -6094.217} C_VEL
LIN {X 0,Y 497.998,Z 324.5,A -85,B 0,C 180,E1 -6094.493,E2 -6094.493} C_VEL
LIN {X 0,Y 498.551,Z 236.33,A -85,B 0,C 180,E1 -6095.815,E2 -6095.815} C_VEL
LIN {X 0,Y 496.323,Z 224.801,A -85,B 0,C 180,E1 -6096.088,E2 -6096.088} C_VEL
LIN {X 0,Y 496.284,Z 210.765,A -85,B 0,C 180,E1 -6098.614,E2 -6098.614} C_VEL
LIN {X 0,Y 495.825,Z 207.726,A -85,B 0,C 180,E1 -6099.192,E2 -6099.192} C_VEL
LIN {X 0,Y 495.751,Z 207.73,A -85,B 0,C 180,E1 -6102.68,E2 -6102.68} C_VEL
LIN {X 0,Y 495.744,Z 207.737,A -85,B 0,C 180,E1 -6105.216,E2 -6105.216} C_VEL
LIN {X 0,Y 495.828,Z 207.723,A -85,B 0,C 180,E1 -6108.555,E2 -6108.555} C_VEL
LIN {X 0,Y 495.824,Z 207.722,A -85,B 0,C 180,E1 -6111.852,E2 -6111.852} C_VEL
LIN {X 0,Y 495.866,Z 207.715,A -85,B 0,C 180,E1 -6114.306,E2 -6114.306} C_VEL
LIN {X 0,Y 495.939,Z 207.708,A -85,B 0,C 180,E1 -6117.564,E2 -6117.564} C_VEL
LIN {X 0,Y 495.939,Z 207.705,A -85,B 0,C 180,E1 -6120,E2 -6120} C_VEL
LIN {X 0,Y 495.938,Z 207.707,A -85,B 0,C 180,E1 -6122.437,E2 -6122.437} C_VEL
LIN {X 0,Y 495.835,Z 207.717,A -85,B 0,C 180,E1 -6125.694,E2 -6125.694} C_VEL
LIN {X 0,Y 495.821,Z 207.719,A -85,B 0,C 180,E1 -6128.149,E2 -6128.149} C_VEL
LIN {X 0,Y 495.822,Z 207.719,A -85,B 0,C 180,E1 -6131.446,E2 -6131.446} C_VEL
LIN {X 0,Y 495.739,Z 207.735,A -85,B 0,C 180,E1 -6134.785,E2 -6134.785} C_VEL
LIN {X 0,Y 495.746,Z 207.729,A -85,B 0,C 180,E1 -6137.32,E2 -6137.32} C_VEL
LIN {X 0,Y 495.724,Z 207.731,A -85,B 0,C 180,E1 -6139.893,E2 -6139.893} C_VEL
LIN {X 0,Y 495.72,Z 207.735,A -85,B 0,C 180,E1 -6142.864,E2 -6142.864} C_VEL
LIN {X 0,Y 495.748,Z 207.73,A -85,B 0,C 180,E1 -6146.071,E2 -6146.071} C_VEL
LIN {X 0,Y 495.731,Z 207.733,A -85,B 0,C 180,E1 -6148.818,E2 -6148.818} C_VEL
LIN {X 0,Y 495.719,Z 207.732,A -85,B 0,C 180,E1 -6151.729,E2 -6151.729} C_VEL
LIN {X 0,Y 495.739,Z 207.732,A -85,B 0,C 180,E1 -6154.698,E2 -6154.698} C_VEL
LIN {X 0,Y 495.697,Z 207.735,A -85,B 0,C 180,E1 -6157.565,E2 -6157.565} C_VEL
LIN {X 0,Y 495.737,Z 207.733,A -85,B 0,C 180,E1 -6160.703,E2 -6160.703} C_VEL
LIN {X 0,Y 495.701,Z 207.738,A -85,B 0,C 180,E1 -6164.005,E2 -6164.005} C_VEL
LIN {X 0,Y 495.702,Z 207.734,A -85,B 0,C 180,E1 -6167.12,E2 -6167.12} C_VEL
LIN {X 0,Y 495.738,Z 207.735,A -85,B 0,C 180,E1 -6169.956,E2 -6169.956} C_VEL
LIN {X 0,Y 495.711,Z 207.736,A -85,B 0,C 180,E1 -6172.556,E2 -6172.556} C_VEL
LIN {X 0,Y 495.768,Z 207.728,A -85,B 0,C 180,E1 -6175.46,E2 -6175.46} C_VEL
LIN {X 0,Y 495.742,Z 207.734,A -85,B 0,C 180,E1 -6178.367,E2 -6178.367} C_VEL
LIN {X 0,Y 495.777,Z 207.732,A -85,B 0,C 180,E1 -6181.51,E2 -6181.51} C_VEL
LIN {X 0,Y 495.838,Z 207.848,A -85,B 0,C 180,E1 -6184.614,E2 -6184.614} C_VEL
LIN {X 0,Y 497.485,Z 217.71,A -85,B 0,C 180,E1 -6186.261,E2 -6186.261} C_VEL
LIN {X 0,Y 497.035,Z 234.824,A -85,B 0,C 180,E1 -6188.945,E2 -6188.945} C_VEL
LIN {X 0,Y 496.468,Z 256.382,A -85,B 0,C 180,E1 -6192.283,E2 -6192.283} C_VEL
LIN {X 0,Y 496.159,Z 267.249,A -85,B 0,C 180,E1 -6193.954,E2 -6193.954} C_VEL
LIN {X 0,Y 498.437,Z 284.18,A -85,B 0,C 180,E1 -6194.289,E2 -6194.289} C_VEL
LIN {X 0,Y 497.828,Z 377.106,A -85,B 0,C 180,E1 -6195.698,E2 -6195.698} C_VEL
LIN {X 0,Y 497.497,Z 390.779,A -85,B 0,C 180,E1 -6196.08,E2 -6196.08} C_VEL
LIN {X 0,Y 497.134,Z 403.634,A -85,B 0,C 180,E1 -6196.616,E2 -6196.616} C_VEL
LIN {X 0,Y 496.764,Z 415.872,A -85,B 0,C 180,E1 -6197.312,E2 -6197.312} C_VEL
LIN {X 0,Y 496.348,Z 427.454,A -85,B 0,C 180,E1 -6198.154,E2 -6198.154} C_VEL
LIN {X 0,Y 496.022,Z 436.557,A -85,B 0,C 180,E1 -6198.974,E2 -6198.974} C_VEL
LIN {X 0,Y 495.722,Z 445.902,A -85,B 0,C 180,E1 -6200,E2 -6200} C_VEL
LIN {X 0,Y 495.44,Z 454.983,A -85,B 0,C 180,E1 -6201.229,E2 -6201.229} C_VEL
LIN {X 0,Y 495.243,Z 462.302,A -85,B 0,C 180,E1 -6202.458,E2 -6202.458} C_VEL
LIN {X 0,Y 495.107,Z 468.521,A -85,B 0,C 180,E1 -6203.777,E2 -6203.777} C_VEL
LIN {X 0,Y 495.034,Z 473.384,A -85,B 0,C 180,E1 -6205.114,E2 -6205.114} C_VEL
LIN {X 0,Y 495.054,Z 475.721,A -85,B 0,C 180,E1 -6205.93,E2 -6205.93} C_VEL
LIN {X 0,Y 495.045,Z 477.619,A -85,B 0,C 180,E1 -6206.745,E2 -6206.745} C_VEL
LIN {X 0,Y 495.025,Z 479.043,A -85,B 0,C 180,E1 -6207.559,E2 -6207.559} C_VEL
LIN {X 0,Y 494.916,Z 480.682,A -85,B 0,C 180,E1 -6209.186,E2 -6209.186} C_VEL
LIN {X 0,Y 494.909,Z 480.909,A -85,B 0,C 180,E1 -6210,E2 -6210} C_VEL
LIN {X 0,Y 494.963,Z 480.092,A -85,B 0,C 180,E1 -6211.627,E2 -6211.627} C_VEL
LIN {X 0,Y 495.024,Z 479.095,A -85,B 0,C 180,E1 -6212.441,E2 -6212.441} C_VEL
LIN {X 0,Y 495.042,Z 477.687,A -85,B 0,C 180,E1 -6213.255,E2 -6213.255} C_VEL
LIN {X 0,Y 495.007,Z 474.723,A -85,B 0,C 180,E1 -6214.478,E2 -6214.478} C_VEL
LIN {X 0,Y 495.115,Z 470.713,A -85,B 0,C 180,E1 -6215.702,E2 -6215.702} C_VEL
LIN {X 0,Y 495.239,Z 464.532,A -85,B 0,C 180,E1 -6217.132,E2 -6217.132} C_VEL
LIN {X 0,Y 495.413,Z 457.783,A -85,B 0,C 180,E1 -6218.36,E2 -6218.36} C_VEL
LIN {X 0,Y 495.63,Z 449.407,A -85,B 0,C 180,E1 -6219.59,E2 -6219.59} C_VEL
LIN {X 0,Y 495.946,Z 440.794,A -85,B 0,C 180,E1 -6220.614,E2 -6220.614} C_VEL
LIN {X 0,Y 496.346,Z 430.168,A -85,B 0,C 180,E1 -6221.639,E2 -6221.639} C_VEL
LIN {X 0,Y 496.69,Z 419.213,A -85,B 0,C 180,E1 -6222.491,E2 -6222.491} C_VEL
LIN {X 0,Y 497.012,Z 408.027,A -85,B 0,C 180,E1 -6223.179,E2 -6223.179} C_VEL
LIN {X 0,Y 497.338,Z 395.985,A -85,B 0,C 180,E1 -6223.742,E2 -6223.742} C_VEL
LIN {X 0,Y 497.693,Z 382.977,A -85,B 0,C 180,E1 -6224.175,E2 -6224.175} C_VEL
LIN {X 0,Y 497.939,Z 370.786,A -85,B 0,C 180,E1 -6224.429,E2 -6224.429} C_VEL
LIN {X 0,Y 498.404,Z 282.556,A -85,B 0,C 180,E1 -6225.74,E2 -6225.74} C_VEL
LIN {X 0,Y 496.233,Z 267.953,A -85,B 0,C 180,E1 -6226.035,E2 -6226.035} C_VEL
LIN {X 0,Y 496.834,Z 247.887,A -85,B 0,C 180,E1 -6229.199,E2 -6229.199} C_VEL
LIN {X 0,Y 497.498,Z 227.745,A -85,B 0,C 180,E1 -6232.419,E2 -6232.419} C_VEL
LIN {X 0,Y 497.822,Z 218.335,A -85,B 0,C 180,E1 -6233.943,E2 -6233.943} C_VEL
LIN {X 0,Y 495.835,Z 207.724,A -85,B 0,C 180,E1 -6235.808,E2 -6235.808} C_VEL
LIN {X 0,Y 495.76,Z 207.73,A -85,B 0,C 180,E1 -6238.812,E2 -6238.812} C_VEL
LIN {X 0,Y 495.742,Z 207.734,A -85,B 0,C 180,E1 -6241.722,E2 -6241.722} C_VEL
LIN {X 0,Y 495.758,Z 207.727,A -85,B 0,C 180,E1 -6244.692,E2 -6244.692} C_VEL
LIN {X 0,Y 495.712,Z 207.736,A -85,B 0,C 180,E1 -6247.558,E2 -6247.558} C_VEL
LIN {X 0,Y 495.745,Z 207.728,A -85,B 0,C 180,E1 -6250.696,E2 -6250.696} C_VEL
LIN {X 0,Y 495.708,Z 207.739,A -85,B 0,C 180,E1 -6253.998,E2 -6253.998} C_VEL
LIN {X 0,Y 495.698,Z 207.735,A -85,B 0,C 180,E1 -6257.113,E2 -6257.113} C_VEL
LIN {X 0,Y 495.727,Z 207.735,A -85,B 0,C 180,E1 -6259.95,E2 -6259.95} C_VEL
LIN {X 0,Y 495.695,Z 207.734,A -85,B 0,C 180,E1 -6262.55,E2 -6262.55} C_VEL
LIN {X 0,Y 495.748,Z 207.734,A -85,B 0,C 180,E1 -6265.454,E2 -6265.454} C_VEL
LIN {X 0,Y 495.719,Z 207.731,A -85,B 0,C 180,E1 -6268.361,E2 -6268.361} C_VEL
LIN {X 0,Y 495.746,Z 207.736,A -85,B 0,C 180,E1 -6271.504,E2 -6271.504} C_VEL
LIN {X 0,Y 495.747,Z 207.73,A -85,B 0,C 180,E1 -6273.929,E2 -6273.929} C_VEL
LIN {X 0,Y 495.719,Z 207.736,A -85,B 0,C 180,E1 -6277.136,E2 -6277.136} C_VEL
LIN {X 0,Y 495.723,Z 207.731,A -85,B 0,C 180,E1 -6280.107,E2 -6280.107} C_VEL
LIN {X 0,Y 495.745,Z 207.729,A -85,B 0,C 180,E1 -6282.68,E2 -6282.68} C_VEL
LIN {X 0,Y 495.738,Z 207.738,A -85,B 0,C 180,E1 -6285.215,E2 -6285.215} C_VEL
LIN {X 0,Y 495.821,Z 207.72,A -85,B 0,C 180,E1 -6288.554,E2 -6288.554} C_VEL
LIN {X 0,Y 495.82,Z 207.719,A -85,B 0,C 180,E1 -6291.851,E2 -6291.851} C_VEL
LIN {X 0,Y 495.835,Z 207.717,A -85,B 0,C 180,E1 -6294.306,E2 -6294.306} C_VEL
LIN {X 0,Y 495.937,Z 207.706,A -85,B 0,C 180,E1 -6297.563,E2 -6297.563} C_VEL
LIN {X 0,Y 495.938,Z 207.704,A -85,B 0,C 180,E1 -6300,E2 -6300} C_VEL
LIN {X 0,Y 495.938,Z 207.707,A -85,B 0,C 180,E1 -6302.436,E2 -6302.436} C_VEL
LIN {X 0,Y 495.865,Z 207.713,A -85,B 0,C 180,E1 -6305.694,E2 -6305.694} C_VEL
LIN {X 0,Y 495.822,Z 207.72,A -85,B 0,C 180,E1 -6308.148,E2 -6308.148} C_VEL
LIN {X 0,Y 495.827,Z 207.718,A -85,B 0,C 180,E1 -6311.445,E2 -6311.445} C_VEL
LIN {X 0,Y 495.743,Z 207.735,A -85,B 0,C 180,E1 -6314.784,E2 -6314.784} C_VEL
LIN {X 0,Y 495.745,Z 207.729,A -85,B 0,C 180,E1 -6317.32,E2 -6317.32} C_VEL
LIN {X 0,Y 495.774,Z 207.731,A -85,B 0,C 180,E1 -6320.691,E2 -6320.691} C_VEL
LIN {X 0,Y 495.733,Z 207.73,A -85,B 0,C 180,E1 -6323.388,E2 -6323.388} C_VEL
LIN {X 0,Y 495.789,Z 207.726,A -85,B 0,C 180,E1 -6326.754,E2 -6326.754} C_VEL
LIN {X 0,Y 495.739,Z 207.73,A -85,B 0,C 180,E1 -6329.748,E2 -6329.748} C_VEL
LIN {X 0,Y 495.753,Z 207.727,A -85,B 0,C 180,E1 -6333.247,E2 -6333.247} C_VEL
LIN {X 0,Y 495.691,Z 207.741,A -85,B 0,C 180,E1 -6336.093,E2 -6336.093} C_VEL
LIN {X 0,Y 495.748,Z 207.729,A -85,B 0,C 180,E1 -6338.774,E2 -6338.774} C_VEL
LIN {X 0,Y 495.753,Z 207.731,A -85,B 0,C 180,E1 -6341.781,E2 -6341.781} C_VEL
LIN {X 0,Y 495.719,Z 207.731,A -85,B 0,C 180,E1 -6345.143,E2 -6345.143} C_VEL
LIN {X 0,Y 495.735,Z 207.735,A -85,B 0,C 180,E1 -6348.222,E2 -6348.222} C_VEL
LIN {X 0,Y 495.745,Z 207.729,A -85,B 0,C 180,E1 -6351.234,E2 -6351.234} C_VEL
LIN {X 0,Y 495.737,Z 207.73,A -85,B 0,C 180,E1 -6354.466,E2 -6354.466} C_VEL
LIN {X 0,Y 495.752,Z 207.73,A -85,B 0,C 180,E1 -6357.409,E2 -6357.409} C_VEL
LIN {X 0,Y 495.766,Z 207.728,A -85,B 0,C 180,E1 -6360.257,E2 -6360.257} C_VEL
LIN {X 0,Y 495.749,Z 207.727,A -85,B 0,C 180,E1 -6360.805,E2 -6360.805} C_VEL
LIN {X 0,Y 495.091,Z 207.816,A -85,B 0,C 180,E1 -6361.484,E2 -6361.484} C_VEL
LIN {X 0,Y 492.234,Z 208.166,A -85,B 0,C 180,E1 -6362.587,E2 -6362.587} C_VEL
LIN {X 0,Y 489.825,Z 208.471,A -85,B 0,C 180,E1 -6363.475,E2 -6363.475} C_VEL
LIN {X 0,Y 488.809,Z 208.594,A -85,B 0,C 180,E1 -6364.162,E2 -6364.162} C_VEL
LIN {X 0,Y 488.737,Z 208.601,A -85,B 0,C 180,E1 -6364.394,E2 -6364.394} C_VEL
LIN {X 0,Y 488.718,Z 208.606,A -85,B 0,C 180,E1 -6367.156,E2 -6367.156} C_VEL
LIN {X 0,Y 488.717,Z 208.609,A -85,B 0,C 180,E1 -6369.813,E2 -6369.813} C_VEL
LIN {X 0,Y 488.727,Z 208.602,A -85,B 0,C 180,E1 -6372.425,E2 -6372.425} C_VEL
LIN {X 0,Y 488.76,Z 208.6,A -85,B 0,C 180,E1 -6375.001,E2 -6375.001} C_VEL
LIN {X 0,Y 488.802,Z 208.593,A -85,B 0,C 180,E1 -6378.389,E2 -6378.389} C_VEL
LIN {X 0,Y 488.815,Z 208.595,A -85,B 0,C 180,E1 -6381.735,E2 -6381.735} C_VEL
LIN {X 0,Y 488.846,Z 208.587,A -85,B 0,C 180,E1 -6384.225,E2 -6384.225} C_VEL
LIN {X 0,Y 488.96,Z 208.578,A -85,B 0,C 180,E1 -6387.529,E2 -6387.529} C_VEL
LIN {X 0,Y 488.969,Z 208.572,A -85,B 0,C 180,E1 -6390,E2 -6390} C_VEL
LIN {X 0,Y 488.96,Z 208.574,A -85,B 0,C 180,E1 -6392.471,E2 -6392.471} C_VEL
LIN {X 0,Y 488.842,Z 208.589,A -85,B 0,C 180,E1 -6395.775,E2 -6395.775} C_VEL
LIN {X 0,Y 488.815,Z 208.592,A -85,B 0,C 180,E1 -6398.266,E2 -6398.266} C_VEL
LIN {X 0,Y 488.802,Z 208.594,A -85,B 0,C 180,E1 -6401.611,E2 -6401.611} C_VEL
LIN {X 0,Y 488.757,Z 208.606,A -85,B 0,C 180,E1 -6404.999,E2 -6404.999} C_VEL
LIN {X 0,Y 488.749,Z 208.603,A -85,B 0,C 180,E1 -6408.44,E2 -6408.44} C_VEL
LIN {X 0,Y 488.7,Z 208.61,A -85,B 0,C 180,E1 -6411.069,E2 -6411.069} C_VEL
LIN {X 0,Y 488.684,Z 208.608,A -85,B 0,C 180,E1 -6413.743,E2 -6413.743} C_VEL
LIN {X 0,Y 488.787,Z 208.602,A -85,B 0,C 180,E1 -6416.943,E2 -6416.943} C_VEL
LIN {X 0,Y 488.807,Z 208.664,A -85,B 0,C 180,E1 -6420.41,E2 -6420.41} C_VEL
LIN {X 0,Y 489.528,Z 214.283,A -85,B 0,C 180,E1 -6421.598,E2 -6421.598} C_VEL
LIN {X 0,Y 489.308,Z 225.178,A -85,B 0,C 180,E1 -6423.802,E2 -6423.802} C_VEL
LIN {X 0,Y 491.736,Z 237.824,A -85,B 0,C 180,E1 -6424.088,E2 -6424.088} C_VEL
LIN {X 0,Y 491.039,Z 331.878,A -85,B 0,C 180,E1 -6425.526,E2 -6425.526} C_VEL
LIN {X 0,Y 490.763,Z 345.075,A -85,B 0,C 180,E1 -6425.887,E2 -6425.887} C_VEL
LIN {X 0,Y 490.571,Z 358.163,A -85,B 0,C 180,E1 -6426.428,E2 -6426.428} C_VEL
LIN {X 0,Y 490.182,Z 369.896,A -85,B 0,C 180,E1 -6427.086,E2 -6427.086} C_VEL
LIN {X 0,Y 489.76,Z 381.912,A -85,B 0,C 180,E1 -6427.959,E2 -6427.959} C_VEL
LIN {X 0,Y 489.403,Z 392.112,A -85,B 0,C 180,E1 -6428.89,E2 -6428.89} C_VEL
LIN {X 0,Y 489.026,Z 402.023,A -85,B 0,C 180,E1 -6430.02,E2 -6430.02} C_VEL
LIN {X 0,Y 488.701,Z 410.019,A -85,B 0,C 180,E1 -6431.139,E2 -6431.139} C_VEL
LIN {X 0,Y 488.405,Z 416.782,A -85,B 0,C 180,E1 -6432.296,E2 -6432.296} C_VEL
LIN {X 0,Y 488.22,Z 423.317,A -85,B 0,C 180,E1 -6433.701,E2 -6433.701} C_VEL
LIN {X 0,Y 488.071,Z 428.334,A -85,B 0,C 180,E1 -6435.124,E2 -6435.124} C_VEL
LIN {X 0,Y 487.991,Z 431.369,A -85,B 0,C 180,E1 -6436.268,E2 -6436.268} C_VEL
LIN {X 0,Y 487.922,Z 433.544,A -85,B 0,C 180,E1 -6437.392,E2 -6437.392} C_VEL
LIN {X 0,Y 487.896,Z 434.898,A -85,B 0,C 180,E1 -6438.501,E2 -6438.501} C_VEL
LIN {X 0,Y 487.849,Z 435.586,A -85,B 0,C 180,E1 -6439.768,E2 -6439.768} C_VEL
LIN {X 0,Y 487.83,Z 435.322,A -85,B 0,C 180,E1 -6441.066,E2 -6441.066} C_VEL
LIN {X 0,Y 487.87,Z 433.494,A -85,B 0,C 180,E1 -6442.769,E2 -6442.769} C_VEL
LIN {X 0,Y 488.017,Z 430.257,A -85,B 0,C 180,E1 -6444.321,E2 -6444.321} C_VEL
LIN {X 0,Y 488.115,Z 425.606,A -85,B 0,C 180,E1 -6445.839,E2 -6445.839} C_VEL
LIN {X 0,Y 488.333,Z 420.45,A -85,B 0,C 180,E1 -6447.092,E2 -6447.092} C_VEL
LIN {X 0,Y 488.6,Z 413.336,A -85,B 0,C 180,E1 -6448.449,E2 -6448.449} C_VEL
LIN {X 0,Y 488.894,Z 405.911,A -85,B 0,C 180,E1 -6449.59,E2 -6449.59} C_VEL
LIN {X 0,Y 489.273,Z 396.487,A -85,B 0,C 180,E1 -6450.766,E2 -6450.766} C_VEL
LIN {X 0,Y 489.595,Z 386.953,A -85,B 0,C 180,E1 -6451.725,E2 -6451.725} C_VEL
LIN {X 0,Y 490.003,Z 375.117,A -85,B 0,C 180,E1 -6452.68,E2 -6452.68} C_VEL
LIN {X 0,Y 490.464,Z 363.662,A -85,B 0,C 180,E1 -6453.398,E2 -6453.398} C_VEL
LIN {X 0,Y 490.758,Z 352.053,A -85,B 0,C 180,E1 -6453.955,E2 -6453.955} C_VEL
LIN {X 0,Y 490.966,Z 339.079,A -85,B 0,C 180,E1 -6454.402,E2 -6454.402} C_VEL
LIN {X 0,Y 491.149,Z 326.077,A -85,B 0,C 180,E1 -6454.678,E2 -6454.678} C_VEL
LIN {X 0,Y 491.781,Z 237.419,A -85,B 0,C 180,E1 -6456.033,E2 -6456.033} C_VEL
LIN {X 0,Y 489.39,Z 225.107,A -85,B 0,C 180,E1 -6456.333,E2 -6456.333} C_VEL
LIN {X 0,Y 489.379,Z 212.998,A -85,B 0,C 180,E1 -6458.518,E2 -6458.518} C_VEL
LIN {X 0,Y 488.755,Z 208.607,A -85,B 0,C 180,E1 -6459.353,E2 -6459.353} C_VEL
LIN {X 0,Y 488.699,Z 208.608,A -85,B 0,C 180,E1 -6462.422,E2 -6462.422} C_VEL
LIN {X 0,Y 488.715,Z 208.611,A -85,B 0,C 180,E1 -6464.998,E2 -6464.998} C_VEL
LIN {X 0,Y 488.785,Z 208.6,A -85,B 0,C 180,E1 -6468.387,E2 -6468.387} C_VEL
LIN {X 0,Y 488.768,Z 208.602,A -85,B 0,C 180,E1 -6471.733,E2 -6471.733} C_VEL
LIN {X 0,Y 488.824,Z 208.592,A -85,B 0,C 180,E1 -6474.224,E2 -6474.224} C_VEL
LIN {X 0,Y 488.907,Z 208.585,A -85,B 0,C 180,E1 -6477.529,E2 -6477.529} C_VEL
LIN {X 0,Y 488.911,Z 208.581,A -85,B 0,C 180,E1 -6480,E2 -6480} C_VEL
LIN {X 0,Y 488.906,Z 208.583,A -85,B 0,C 180,E1 -6482.472,E2 -6482.472} C_VEL
LIN {X 0,Y 488.794,Z 208.593,A -85,B 0,C 180,E1 -6485.777,E2 -6485.777} C_VEL
LIN {X 0,Y 488.766,Z 208.599,A -85,B 0,C 180,E1 -6488.268,E2 -6488.268} C_VEL
LIN {X 0,Y 488.782,Z 208.595,A -85,B 0,C 180,E1 -6491.613,E2 -6491.613} C_VEL
LIN {X 0,Y 488.711,Z 208.61,A -85,B 0,C 180,E1 -6495.002,E2 -6495.002} C_VEL
LIN {X 0,Y 488.713,Z 208.607,A -85,B 0,C 180,E1 -6498.374,E2 -6498.374} C_VEL
LIN {X 0,Y 488.666,Z 208.614,A -85,B 0,C 180,E1 -6501.073,E2 -6501.073} C_VEL
LIN {X 0,Y 488.655,Z 208.609,A -85,B 0,C 180,E1 -6503.748,E2 -6503.748} C_VEL
LIN {X 0,Y 488.75,Z 208.603,A -85,B 0,C 180,E1 -6506.946,E2 -6506.946} C_VEL
LIN {X 0,Y 488.67,Z 208.614,A -85,B 0,C 180,E1 -6510.366,E2 -6510.366} C_VEL
LIN {X 0,Y 488.699,Z 208.606,A -85,B 0,C 180,E1 -6513.487,E2 -6513.487} C_VEL
LIN {X 0,Y 488.654,Z 208.618,A -85,B 0,C 180,E1 -6516.359,E2 -6516.359} C_VEL
LIN {X 0,Y 488.669,Z 208.611,A -85,B 0,C 180,E1 -6519.258,E2 -6519.258} C_VEL
LIN {X 0,Y 488.679,Z 208.61,A -85,B 0,C 180,E1 -6521.603,E2 -6521.603} C_VEL
LIN {X 0,Y 488.675,Z 208.61,A -85,B 0,C 180,E1 -6524.806,E2 -6524.806} C_VEL
LIN {X 0,Y 488.668,Z 208.611,A -85,B 0,C 180,E1 -6527.478,E2 -6527.478} C_VEL
LIN {X 0,Y 488.713,Z 208.608,A -85,B 0,C 180,E1 -6529.68,E2 -6529.68} C_VEL
LIN {X 0,Y 488.664,Z 208.612,A -85,B 0,C 180,E1 -6532.844,E2 -6532.844} C_VEL
LIN {X 0,Y 488.719,Z 208.611,A -85,B 0,C 180,E1 -6535.89,E2 -6535.89} C_VEL
LIN {X 0,Y 488.679,Z 208.611,A -85,B 0,C 180,E1 -6538.823,E2 -6538.823} C_VEL
LIN {X 0,Y 488.734,Z 208.61,A -85,B 0,C 180,E1 -6541.674,E2 -6541.674} C_VEL
LIN {X 0,Y 488.801,Z 208.681,A -85,B 0,C 180,E1 -6544.422,E2 -6544.422} C_VEL
LIN {X 0,Y 490.544,Z 218.728,A -85,B 0,C 180,E1 -6546.128,E2 -6546.128} C_VEL
LIN {X 0,Y 490.089,Z 235.321,A -85,B 0,C 180,E1 -6548.768,E2 -6548.768} C_VEL
LIN {X 0,Y 489.447,Z 257.417,A -85,B 0,C 180,E1 -6552.236,E2 -6552.236} C_VEL
LIN {X 0,Y 489.183,Z 266.881,A -85,B 0,C 180,E1 -6553.712,E2 -6553.712} C_VEL
LIN {X 0,Y 491.623,Z 284.037,A -85,B 0,C 180,E1 -6554.066,E2 -6554.066} C_VEL
LIN {X 0,Y 490.939,Z 376.627,A -85,B 0,C 180,E1 -6555.493,E2 -6555.493} C_VEL
LIN {X 0,Y 490.642,Z 389.563,A -85,B 0,C 180,E1 -6555.855,E2 -6555.855} C_VEL
LIN {X 0,Y 490.229,Z 402.161,A -85,B 0,C 180,E1 -6556.372,E2 -6556.372} C_VEL
LIN {X 0,Y 489.801,Z 414.676,A -85,B 0,C 180,E1 -6557.077,E2 -6557.077} C_VEL
LIN {X 0,Y 489.422,Z 425.739,A -85,B 0,C 180,E1 -6557.878,E2 -6557.878} C_VEL
LIN {X 0,Y 489.048,Z 436.156,A -85,B 0,C 180,E1 -6558.815,E2 -6558.815} C_VEL
LIN {X 0,Y 488.684,Z 445.513,A -85,B 0,C 180,E1 -6559.854,E2 -6559.854} C_VEL
LIN {X 0,Y 488.391,Z 454.609,A -85,B 0,C 180,E1 -6561.102,E2 -6561.102} C_VEL
LIN {X 0,Y 488.178,Z 461.939,A -85,B 0,C 180,E1 -6562.348,E2 -6562.348} C_VEL
LIN {X 0,Y 488.043,Z 467.528,A -85,B 0,C 180,E1 -6563.53,E2 -6563.53} C_VEL
LIN {X 0,Y 488.01,Z 471.701,A -85,B 0,C 180,E1 -6564.629,E2 -6564.629} C_VEL
LIN {X 0,Y 487.947,Z 475.38,A -85,B 0,C 180,E1 -6565.871,E2 -6565.871} C_VEL
LIN {X 0,Y 487.969,Z 477.284,A -85,B 0,C 180,E1 -6566.698,E2 -6566.698} C_VEL
LIN {X 0,Y 487.933,Z 478.71,A -85,B 0,C 180,E1 -6567.524,E2 -6567.524} C_VEL
LIN {X 0,Y 487.892,Z 479.729,A -85,B 0,C 180,E1 -6568.349,E2 -6568.349} C_VEL
LIN {X 0,Y 487.829,Z 480.583,A -85,B 0,C 180,E1 -6570,E2 -6570} C_VEL
LIN {X 0,Y 487.892,Z 479.768,A -85,B 0,C 180,E1 -6571.651,E2 -6571.651} C_VEL
LIN {X 0,Y 487.933,Z 478.769,A -85,B 0,C 180,E1 -6572.476,E2 -6572.476} C_VEL
LIN {X 0,Y 487.965,Z 477.359,A -85,B 0,C 180,E1 -6573.302,E2 -6573.302} C_VEL
LIN {X 0,Y 487.919,Z 474.392,A -85,B 0,C 180,E1 -6574.543,E2 -6574.543} C_VEL
LIN {X 0,Y 488.01,Z 470.375,A -85,B 0,C 180,E1 -6575.785,E2 -6575.785} C_VEL
LIN {X 0,Y 488.171,Z 464.185,A -85,B 0,C 180,E1 -6577.236,E2 -6577.236} C_VEL
LIN {X 0,Y 488.344,Z 457.426,A -85,B 0,C 180,E1 -6578.482,E2 -6578.482} C_VEL
LIN {X 0,Y 488.569,Z 449.036,A -85,B 0,C 180,E1 -6579.73,E2 -6579.73} C_VEL
LIN {X 0,Y 488.919,Z 440.403,A -85,B 0,C 180,E1 -6580.769,E2 -6580.769} C_VEL
LIN {X 0,Y 489.348,Z 429.76,A -85,B 0,C 180,E1 -6581.808,E2 -6581.808} C_VEL
LIN {X 0,Y 489.696,Z 419.79,A -85,B 0,C 180,E1 -6582.598,E2 -6582.598} C_VEL
LIN {X 0,Y 490.091,Z 407.559,A -85,B 0,C 180,E1 -6583.368,E2 -6583.368} C_VEL
LIN {X 0,Y 490.454,Z 395.472,A -85,B 0,C 180,E1 -6583.939,E2 -6583.939} C_VEL
LIN {X 0,Y 490.815,Z 382.392,A -85,B 0,C 180,E1 -6584.378,E2 -6584.378} C_VEL
LIN {X 0,Y 491.055,Z 369.992,A -85,B 0,C 180,E1 -6584.635,E2 -6584.635} C_VEL
LIN {X 0,Y 491.501,Z 282.82,A -85,B 0,C 180,E1 -6585.955,E2 -6585.955} C_VEL
LIN {X 0,Y 489.246,Z 267.671,A -85,B 0,C 180,E1 -6586.266,E2 -6586.266} C_VEL
LIN {X 0,Y 489.879,Z 247.573,A -85,B 0,C 180,E1 -6589.482,E2 -6589.482} C_VEL
LIN {X 0,Y 490.541,Z 228.776,A -85,B 0,C 180,E1 -6592.532,E2 -6592.532} C_VEL
LIN {X 0,Y 490.842,Z 219.377,A -85,B 0,C 180,E1 -6594.081,E2 -6594.081} C_VEL
LIN {X 0,Y 488.762,Z 208.606,A -85,B 0,C 180,E1 -6596.009,E2 -6596.009} C_VEL
LIN {X 0,Y 488.712,Z 208.608,A -85,B 0,C 180,E1 -6599.267,E2 -6599.267} C_VEL
LIN {X 0,Y 488.689,Z 208.615,A -85,B 0,C 180,E1 -6602.144,E2 -6602.144} C_VEL
LIN {X 0,Y 488.705,Z 208.605,A -85,B 0,C 180,E1 -6605.111,E2 -6605.111} C_VEL
LIN {X 0,Y 488.66,Z 208.615,A -85,B 0,C 180,E1 -6608.197,E2 -6608.197} C_VEL
LIN {X 0,Y 488.697,Z 208.608,A -85,B 0,C 180,E1 -6610.341,E2 -6610.341} C_VEL
LIN {X 0,Y 488.661,Z 208.617,A -85,B 0,C 180,E1 -6613.651,E2 -6613.651} C_VEL
LIN {X 0,Y 488.659,Z 208.612,A -85,B 0,C 180,E1 -6616.342,E2 -6616.342} C_VEL
LIN {X 0,Y 488.703,Z 208.614,A -85,B 0,C 180,E1 -6619.673,E2 -6619.673} C_VEL
LIN {X 0,Y 488.647,Z 208.612,A -85,B 0,C 180,E1 -6622.838,E2 -6622.838} C_VEL
LIN {X 0,Y 488.698,Z 208.61,A -85,B 0,C 180,E1 -6625.884,E2 -6625.884} C_VEL
LIN {X 0,Y 488.654,Z 208.612,A -85,B 0,C 180,E1 -6628.817,E2 -6628.817} C_VEL
LIN {X 0,Y 488.703,Z 208.611,A -85,B 0,C 180,E1 -6631.668,E2 -6631.668} C_VEL
LIN {X 0,Y 488.704,Z 208.605,A -85,B 0,C 180,E1 -6634.442,E2 -6634.442} C_VEL
LIN {X 0,Y 488.681,Z 208.613,A -85,B 0,C 180,E1 -6637.151,E2 -6637.151} C_VEL
LIN {X 0,Y 488.678,Z 208.611,A -85,B 0,C 180,E1 -6639.808,E2 -6639.808} C_VEL
LIN {X 0,Y 488.69,Z 208.607,A -85,B 0,C 180,E1 -6642.421,E2 -6642.421} C_VEL
LIN {X 0,Y 488.71,Z 208.61,A -85,B 0,C 180,E1 -6644.998,E2 -6644.998} C_VEL
LIN {X 0,Y 488.781,Z 208.596,A -85,B 0,C 180,E1 -6648.387,E2 -6648.387} C_VEL
LIN {X 0,Y 488.765,Z 208.599,A -85,B 0,C 180,E1 -6651.732,E2 -6651.732} C_VEL
LIN {X 0,Y 488.793,Z 208.594,A -85,B 0,C 180,E1 -6654.223,E2 -6654.223} C_VEL
LIN {X 0,Y 488.905,Z 208.582,A -85,B 0,C 180,E1 -6657.528,E2 -6657.528} C_VEL
LIN {X 0,Y 488.923,Z 208.585,A -85,B 0,C 180,E1 -6660.823,E2 -6660.823} C_VEL
LIN {X 0,Y 488.906,Z 208.583,A -85,B 0,C 180,E1 -6662.471,E2 -6662.471} C_VEL
LIN {X 0,Y 488.823,Z 208.59,A -85,B 0,C 180,E1 -6665.776,E2 -6665.776} C_VEL
LIN {X 0,Y 488.767,Z 208.599,A -85,B 0,C 180,E1 -6668.267,E2 -6668.267} C_VEL
LIN {X 0,Y 488.784,Z 208.595,A -85,B 0,C 180,E1 -6671.613,E2 -6671.613} C_VEL
LIN {X 0,Y 488.713,Z 208.608,A -85,B 0,C 180,E1 -6675.002,E2 -6675.002} C_VEL
LIN {X 0,Y 488.706,Z 208.611,A -85,B 0,C 180,E1 -6678.444,E2 -6678.444} C_VEL
LIN {X 0,Y 488.717,Z 208.605,A -85,B 0,C 180,E1 -6681.07,E2 -6681.07} C_VEL
LIN {X 0,Y 488.671,Z 208.61,A -85,B 0,C 180,E1 -6683.746,E2 -6683.746} C_VEL
LIN {X 0,Y 488.754,Z 208.601,A -85,B 0,C 180,E1 -6686.947,E2 -6686.947} C_VEL
LIN {X 0,Y 488.677,Z 208.617,A -85,B 0,C 180,E1 -6690.367,E2 -6690.367} C_VEL
LIN {X 0,Y 488.696,Z 208.606,A -85,B 0,C 180,E1 -6693.487,E2 -6693.487} C_VEL
LIN {X 0,Y 488.652,Z 208.618,A -85,B 0,C 180,E1 -6696.358,E2 -6696.358} C_VEL
LIN {X 0,Y 488.721,Z 208.603,A -85,B 0,C 180,E1 -6699.252,E2 -6699.252} C_VEL
LIN {X 0,Y 488.702,Z 208.608,A -85,B 0,C 180,E1 -6702.524,E2 -6702.524} C_VEL
LIN {X 0,Y 488.682,Z 208.608,A -85,B 0,C 180,E1 -6705.202,E2 -6705.202} C_VEL
LIN {X 0,Y 488.687,Z 208.61,A -85,B 0,C 180,E1 -6708.403,E2 -6708.403} C_VEL
LIN {X 0,Y 488.717,Z 208.603,A -85,B 0,C 180,E1 -6710.945,E2 -6710.945} C_VEL
LIN {X 0,Y 488.664,Z 208.618,A -85,B 0,C 180,E1 -6713.872,E2 -6713.872} C_VEL
LIN {X 0,Y 488.721,Z 208.603,A -85,B 0,C 180,E1 -6716.88,E2 -6716.88} C_VEL
LIN {X 0,Y 488.718,Z 208.612,A -85,B 0,C 180,E1 -6719.784,E2 -6719.784} C_VEL
LIN {X 0,Y 488.786,Z 208.596,A -85,B 0,C 180,E1 -6723.057,E2 -6723.057} C_VEL
LIN {X 0,Y 488.737,Z 208.601,A -85,B 0,C 180,E1 -6724.394,E2 -6724.394} C_VEL
LIN {X 0,Y 488.092,Z 208.684,A -85,B 0,C 180,E1 -6725.082,E2 -6725.082} C_VEL
LIN {X 0,Y 485.221,Z 209.047,A -85,B 0,C 180,E1 -6726.198,E2 -6726.198} C_VEL
LIN {X 0,Y 482.773,Z 209.353,A -85,B 0,C 180,E1 -6727.098,E2 -6727.098} C_VEL
LIN {X 0,Y 481.716,Z 209.482,A -85,B 0,C 180,E1 -6727.794,E2 -6727.794} C_VEL
LIN {X 0,Y 481.628,Z 209.49,A -85,B 0,C 180,E1 -6728.03,E2 -6728.03} C_VEL
LIN {X 0,Y 481.698,Z 209.478,A -85,B 0,C 180,E1 -6730.395,E2 -6730.395} C_VEL
LIN {X 0,Y 481.685,Z 209.482,A -85,B 0,C 180,E1 -6733.036,E2 -6733.036} C_VEL
LIN {X 0,Y 481.689,Z 209.485,A -85,B 0,C 180,E1 -6735.64,E2 -6735.64} C_VEL
LIN {X 0,Y 481.747,Z 209.472,A -85,B 0,C 180,E1 -6738.216,E2 -6738.216} C_VEL
LIN {X 0,Y 481.761,Z 209.475,A -85,B 0,C 180,E1 -6741.613,E2 -6741.613} C_VEL
LIN {X 0,Y 481.806,Z 209.465,A -85,B 0,C 180,E1 -6744.14,E2 -6744.14} C_VEL
LIN {X 0,Y 481.927,Z 209.454,A -85,B 0,C 180,E1 -6747.493,E2 -6747.493} C_VEL
LIN {X 0,Y 481.94,Z 209.448,A -85,B 0,C 180,E1 -6750,E2 -6750} C_VEL
LIN {X 0,Y 481.927,Z 209.45,A -85,B 0,C 180,E1 -6752.507,E2 -6752.507} C_VEL
LIN {X 0,Y 481.802,Z 209.465,A -85,B 0,C 180,E1 -6755.86,E2 -6755.86} C_VEL
LIN {X 0,Y 481.761,Z 209.471,A -85,B 0,C 180,E1 -6758.387,E2 -6758.387} C_VEL
LIN {X 0,Y 481.748,Z 209.472,A -85,B 0,C 180,E1 -6761.784,E2 -6761.784} C_VEL
LIN {X 0,Y 481.738,Z 209.477,A -85,B 0,C 180,E1 -6765.223,E2 -6765.223} C_VEL
LIN {X 0,Y 481.706,Z 209.484,A -85,B 0,C 180,E1 -6768.72,E2 -6768.72} C_VEL
LIN {X 0,Y 481.639,Z 209.487,A -85,B 0,C 180,E1 -6771.393,E2 -6771.393} C_VEL
LIN {X 0,Y 481.667,Z 209.483,A -85,B 0,C 180,E1 -6774.111,E2 -6774.111} C_VEL
LIN {X 0,Y 481.74,Z 209.478,A -85,B 0,C 180,E1 -6777.138,E2 -6777.138} C_VEL
LIN {X 0,Y 481.788,Z 209.677,A -85,B 0,C 180,E1 -6780.297,E2 -6780.297} C_VEL
LIN {X 0,Y 482.546,Z 214.71,A -85,B 0,C 180,E1 -6781.374,E2 -6781.374} C_VEL
LIN {X 0,Y 482.357,Z 225.433,A -85,B 0,C 180,E1 -6783.568,E2 -6783.568} C_VEL
LIN {X 0,Y 484.934,Z 238.867,A -85,B 0,C 180,E1 -6783.876,E2 -6783.876} C_VEL
LIN {X 0,Y 484.138,Z 332.503,A -85,B 0,C 180,E1 -6785.333,E2 -6785.333} C_VEL
LIN {X 0,Y 483.876,Z 345.782,A -85,B 0,C 180,E1 -6785.708,E2 -6785.708} C_VEL
LIN {X 0,Y 483.656,Z 358.466,A -85,B 0,C 180,E1 -6786.241,E2 -6786.241} C_VEL
LIN {X 0,Y 483.272,Z 369.863,A -85,B 0,C 180,E1 -6786.886,E2 -6786.886} C_VEL
LIN {X 0,Y 482.858,Z 380.82,A -85,B 0,C 180,E1 -6787.679,E2 -6787.679} C_VEL
LIN {X 0,Y 482.485,Z 391.123,A -85,B 0,C 180,E1 -6788.609,E2 -6788.609} C_VEL
LIN {X 0,Y 482.074,Z 400.349,A -85,B 0,C 180,E1 -6789.629,E2 -6789.629} C_VEL
LIN {X 0,Y 481.772,Z 409.016,A -85,B 0,C 180,E1 -6790.814,E2 -6790.814} C_VEL
LIN {X 0,Y 481.355,Z 417.08,A -85,B 0,C 180,E1 -6792.187,E2 -6792.187} C_VEL
LIN {X 0,Y 481.211,Z 422.496,A -85,B 0,C 180,E1 -6793.342,E2 -6793.342} C_VEL
LIN {X 0,Y 481.089,Z 426.939,A -85,B 0,C 180,E1 -6794.518,E2 -6794.518} C_VEL
LIN {X 0,Y 480.965,Z 430.485,A -85,B 0,C 180,E1 -6795.719,E2 -6795.719} C_VEL
LIN {X 0,Y 480.875,Z 433.148,A -85,B 0,C 180,E1 -6796.943,E2 -6796.943} C_VEL
LIN {X 0,Y 480.798,Z 434.945,A -85,B 0,C 180,E1 -6798.194,E2 -6798.194} C_VEL
LIN {X 0,Y 480.768,Z 435.851,A -85,B 0,C 180,E1 -6799.47,E2 -6799.47} C_VEL
LIN {X 0,Y 480.761,Z 435.666,A -85,B 0,C 180,E1 -6801.054,E2 -6801.054} C_VEL
LIN {X 0,Y 480.754,Z 434.769,A -85,B 0,C 180,E1 -6802.122,E2 -6802.122} C_VEL
LIN {X 0,Y 480.857,Z 432.615,A -85,B 0,C 180,E1 -6803.491,E2 -6803.491} C_VEL
LIN {X 0,Y 480.956,Z 429.187,A -85,B 0,C 180,E1 -6804.906,E2 -6804.906} C_VEL
LIN {X 0,Y 481.133,Z 424.295,A -85,B 0,C 180,E1 -6806.358,E2 -6806.358} C_VEL
LIN {X 0,Y 481.346,Z 418.819,A -85,B 0,C 180,E1 -6807.609,E2 -6807.609} C_VEL
LIN {X 0,Y 481.613,Z 412.349,A -85,B 0,C 180,E1 -6808.8,E2 -6808.8} C_VEL
LIN {X 0,Y 481.987,Z 403.986,A -85,B 0,C 180,E1 -6810.039,E2 -6810.039} C_VEL
LIN {X 0,Y 482.403,Z 394.743,A -85,B 0,C 180,E1 -6811.146,E2 -6811.146} C_VEL
LIN {X 0,Y 482.723,Z 384.852,A -85,B 0,C 180,E1 -6812.115,E2 -6812.115} C_VEL
LIN {X 0,Y 483.136,Z 374.888,A -85,B 0,C 180,E1 -6812.903,E2 -6812.903} C_VEL
LIN {X 0,Y 483.576,Z 363.286,A -85,B 0,C 180,E1 -6813.63,E2 -6813.63} C_VEL
LIN {X 0,Y 483.922,Z 350.522,A -85,B 0,C 180,E1 -6814.233,E2 -6814.233} C_VEL
LIN {X 0,Y 484.156,Z 337.624,A -85,B 0,C 180,E1 -6814.66,E2 -6814.66} C_VEL
LIN {X 0,Y 484.291,Z 323.165,A -85,B 0,C 180,E1 -6814.94,E2 -6814.94} C_VEL
LIN {X 0,Y 484.992,Z 238.325,A -85,B 0,C 180,E1 -6816.259,E2 -6816.259} C_VEL
LIN {X 0,Y 482.451,Z 225.404,A -85,B 0,C 180,E1 -6816.583,E2 -6816.583} C_VEL
LIN {X 0,Y 482.385,Z 213.231,A -85,B 0,C 180,E1 -6818.801,E2 -6818.801} C_VEL
LIN {X 0,Y 481.701,Z 209.486,A -85,B 0,C 180,E1 -6819.559,E2 -6819.559} C_VEL
LIN {X 0,Y 481.677,Z 209.484,A -85,B 0,C 180,E1 -6822.158,E2 -6822.158} C_VEL
LIN {X 0,Y 481.694,Z 209.484,A -85,B 0,C 180,E1 -6824.775,E2 -6824.775} C_VEL
LIN {X 0,Y 481.747,Z 209.477,A -85,B 0,C 180,E1 -6828.215,E2 -6828.215} C_VEL
LIN {X 0,Y 481.714,Z 209.482,A -85,B 0,C 180,E1 -6831.611,E2 -6831.611} C_VEL
LIN {X 0,Y 481.784,Z 209.469,A -85,B 0,C 180,E1 -6834.139,E2 -6834.139} C_VEL
LIN {X 0,Y 481.875,Z 209.461,A -85,B 0,C 180,E1 -6837.493,E2 -6837.493} C_VEL
LIN {X 0,Y 481.854,Z 209.466,A -85,B 0,C 180,E1 -6840.836,E2 -6840.836} C_VEL
LIN {X 0,Y 481.874,Z 209.46,A -85,B 0,C 180,E1 -6842.508,E2 -6842.508} C_VEL
LIN {X 0,Y 481.754,Z 209.47,A -85,B 0,C 180,E1 -6845.861,E2 -6845.861} C_VEL
LIN {X 0,Y 481.712,Z 209.479,A -85,B 0,C 180,E1 -6848.389,E2 -6848.389} C_VEL
LIN {X 0,Y 481.746,Z 209.471,A -85,B 0,C 180,E1 -6851.785,E2 -6851.785} C_VEL
LIN {X 0,Y 481.678,Z 209.481,A -85,B 0,C 180,E1 -6855.661,E2 -6855.661} C_VEL
LIN {X 0,Y 481.666,Z 209.49,A -85,B 0,C 180,E1 -6858.724,E2 -6858.724} C_VEL
LIN {X 0,Y 481.608,Z 209.491,A -85,B 0,C 180,E1 -6861.397,E2 -6861.397} C_VEL
LIN {X 0,Y 481.637,Z 209.486,A -85,B 0,C 180,E1 -6864.116,E2 -6864.116} C_VEL
LIN {X 0,Y 481.706,Z 209.479,A -85,B 0,C 180,E1 -6867.142,E2 -6867.142} C_VEL
LIN {X 0,Y 481.639,Z 209.484,A -85,B 0,C 180,E1 -6869.744,E2 -6869.744} C_VEL
LIN {X 0,Y 481.636,Z 209.491,A -85,B 0,C 180,E1 -6872.677,E2 -6872.677} C_VEL
LIN {X 0,Y 481.608,Z 209.489,A -85,B 0,C 180,E1 -6875.712,E2 -6875.712} C_VEL
LIN {X 0,Y 481.638,Z 209.489,A -85,B 0,C 180,E1 -6878.863,E2 -6878.863} C_VEL
LIN {X 0,Y 481.625,Z 209.491,A -85,B 0,C 180,E1 -6881.916,E2 -6881.916} C_VEL
LIN {X 0,Y 481.629,Z 209.491,A -85,B 0,C 180,E1 -6884.461,E2 -6884.461} C_VEL
LIN {X 0,Y 481.625,Z 209.492,A -85,B 0,C 180,E1 -6887.843,E2 -6887.843} C_VEL
LIN {X 0,Y 481.66,Z 209.486,A -85,B 0,C 180,E1 -6890.655,E2 -6890.655} C_VEL
LIN {X 0,Y 481.613,Z 209.491,A -85,B 0,C 180,E1 -6893.379,E2 -6893.379} C_VEL
LIN {X 0,Y 481.696,Z 209.484,A -85,B 0,C 180,E1 -6896.333,E2 -6896.333} C_VEL
LIN {X 0,Y 481.638,Z 209.49,A -85,B 0,C 180,E1 -6899.421,E2 -6899.421} C_VEL
LIN {X 0,Y 481.69,Z 209.488,A -85,B 0,C 180,E1 -6902.171,E2 -6902.171} C_VEL
LIN {X 0,Y 481.758,Z 209.542,A -85,B 0,C 180,E1 -6904.224,E2 -6904.224} C_VEL
LIN {X 0,Y 483.568,Z 219.764,A -85,B 0,C 180,E1 -6905.99,E2 -6905.99} C_VEL
LIN {X 0,Y 483.138,Z 235.845,A -85,B 0,C 180,E1 -6908.589,E2 -6908.589} C_VEL
LIN {X 0,Y 482.481,Z 257.067,A -85,B 0,C 180,E1 -6911.971,E2 -6911.971} C_VEL
LIN {X 0,Y 482.218,Z 266.493,A -85,B 0,C 180,E1 -6913.461,E2 -6913.461} C_VEL
LIN {X 0,Y 484.795,Z 285.958,A -85,B 0,C 180,E1 -6913.865,E2 -6913.865} C_VEL
LIN {X 0,Y 484.083,Z 376.201,A -85,B 0,C 180,E1 -6915.283,E2 -6915.283} C_VEL
LIN {X 0,Y 483.802,Z 388.382,A -85,B 0,C 180,E1 -6915.624,E2 -6915.624} C_VEL
LIN {X 0,Y 483.375,Z 400.616,A -85,B 0,C 180,E1 -6916.121,E2 -6916.121} C_VEL
LIN {X 0,Y 482.929,Z 412.51,A -85,B 0,C 180,E1 -6916.772,E2 -6916.772} C_VEL
LIN {X 0,Y 482.601,Z 422.871,A -85,B 0,C 180,E1 -6917.501,E2 -6917.501} C_VEL
LIN {X 0,Y 482.16,Z 433.618,A -85,B 0,C 180,E1 -6918.44,E2 -6918.44} C_VEL
LIN {X 0,Y 481.711,Z 443.411,A -85,B 0,C 180,E1 -6919.493,E2 -6919.493} C_VEL
LIN {X 0,Y 481.429,Z 451.449,A -85,B 0,C 180,E1 -6920.548,E2 -6920.548} C_VEL
LIN {X 0,Y 481.159,Z 459.31,A -85,B 0,C 180,E1 -6921.813,E2 -6921.813} C_VEL
LIN {X 0,Y 480.964,Z 466.536,A -85,B 0,C 180,E1 -6923.288,E2 -6923.288} C_VEL
LIN {X 0,Y 480.92,Z 471.356,A -85,B 0,C 180,E1 -6924.55,E2 -6924.55} C_VEL
LIN {X 0,Y 480.844,Z 475.042,A -85,B 0,C 180,E1 -6925.809,E2 -6925.809} C_VEL
LIN {X 0,Y 480.894,Z 476.95,A -85,B 0,C 180,E1 -6926.649,E2 -6926.649} C_VEL
LIN {X 0,Y 480.845,Z 478.379,A -85,B 0,C 180,E1 -6927.487,E2 -6927.487} C_VEL
LIN {X 0,Y 480.823,Z 479.401,A -85,B 0,C 180,E1 -6928.325,E2 -6928.325} C_VEL
LIN {X 0,Y 480.765,Z 480.028,A -85,B 0,C 180,E1 -6929.162,E2 -6929.162} C_VEL
LIN {X 0,Y 480.753,Z 480.257,A -85,B 0,C 180,E1 -6930,E2 -6930} C_VEL
LIN {X 0,Y 480.823,Z 479.441,A -85,B 0,C 180,E1 -6931.675,E2 -6931.675} C_VEL
LIN {X 0,Y 480.845,Z 478.441,A -85,B 0,C 180,E1 -6932.513,E2 -6932.513} C_VEL
LIN {X 0,Y 480.889,Z 477.029,A -85,B 0,C 180,E1 -6933.351,E2 -6933.351} C_VEL
LIN {X 0,Y 480.838,Z 474.058,A -85,B 0,C 180,E1 -6934.61,E2 -6934.61} C_VEL
LIN {X 0,Y 480.915,Z 470.034,A -85,B 0,C 180,E1 -6935.871,E2 -6935.871} C_VEL
LIN {X 0,Y 481.095,Z 463.835,A -85,B 0,C 180,E1 -6937.343,E2 -6937.343} C_VEL
LIN {X 0,Y 481.286,Z 457.066,A -85,B 0,C 180,E1 -6938.607,E2 -6938.607} C_VEL
LIN {X 0,Y 481.525,Z 448.661,A -85,B 0,C 180,E1 -6939.874,E2 -6939.874} C_VEL
LIN {X 0,Y 481.904,Z 440.008,A -85,B 0,C 180,E1 -6940.928,E2 -6940.928} C_VEL
LIN {X 0,Y 482.349,Z 429.451,A -85,B 0,C 180,E1 -6941.972,E2 -6941.972} C_VEL
LIN {X 0,Y 482.752,Z 419.053,A -85,B 0,C 180,E1 -6942.804,E2 -6942.804} C_VEL
LIN {X 0,Y 483.159,Z 407.051,A -85,B 0,C 180,E1 -6943.564,E2 -6943.564} C_VEL
LIN {X 0,Y 483.566,Z 394.903,A -85,B 0,C 180,E1 -6944.142,E2 -6944.142} C_VEL
LIN {X 0,Y 483.932,Z 381.722,A -85,B 0,C 180,E1 -6944.587,E2 -6944.587} C_VEL
LIN {X 0,Y 484.179,Z 369.003,A -85,B 0,C 180,E1 -6944.848,E2 -6944.848} C_VEL
LIN {X 0,Y 484.656,Z 283.566,A -85,B 0,C 180,E1 -6946.164,E2 -6946.164} C_VEL
LIN {X 0,Y 482.25,Z 267.34,A -85,B 0,C 180,E1 -6946.508,E2 -6946.508} C_VEL
LIN {X 0,Y 482.89,Z 248.586,A -85,B 0,C 180,E1 -6949.555,E2 -6949.555} C_VEL
LIN {X 0,Y 483.587,Z 229.808,A -85,B 0,C 180,E1 -6952.649,E2 -6952.649} C_VEL
LIN {X 0,Y 483.956,Z 221.734,A -85,B 0,C 180,E1 -6953.989,E2 -6953.989} C_VEL
LIN {X 0,Y 482.379,Z 212.601,A -85,B 0,C 180,E1 -6955.62,E2 -6955.62} C_VEL
LIN {X 0,Y 481.725,Z 209.483,A -85,B 0,C 180,E1 -6956.214,E2 -6956.214} C_VEL
LIN {X 0,Y 481.666,Z 209.486,A -85,B 0,C 180,E1 -6958.9,E2 -6958.9} C_VEL
LIN {X 0,Y 481.643,Z 209.492,A -85,B 0,C 180,E1 -6962.186,E2 -6962.186} C_VEL
LIN {X 0,Y 481.676,Z 209.481,A -85,B 0,C 180,E1 -6964.679,E2 -6964.679} C_VEL
LIN {X 0,Y 481.636,Z 209.493,A -85,B 0,C 180,E1 -6968.004,E2 -6968.004} C_VEL
LIN {X 0,Y 481.635,Z 209.486,A -85,B 0,C 180,E1 -6971.038,E2 -6971.038} C_VEL
LIN {X 0,Y 481.634,Z 209.487,A -85,B 0,C 180,E1 -6974.454,E2 -6974.454} C_VEL
LIN {X 0,Y 481.619,Z 209.495,A -85,B 0,C 180,E1 -6977.836,E2 -6977.836} C_VEL
LIN {X 0,Y 481.629,Z 209.486,A -85,B 0,C 180,E1 -6980.651,E2 -6980.651} C_VEL
LIN {X 0,Y 481.597,Z 209.495,A -85,B 0,C 180,E1 -6983.372,E2 -6983.372} C_VEL
LIN {X 0,Y 481.674,Z 209.481,A -85,B 0,C 180,E1 -6986.327,E2 -6986.327} C_VEL
LIN {X 0,Y 481.611,Z 209.496,A -85,B 0,C 180,E1 -6989.415,E2 -6989.415} C_VEL
LIN {X 0,Y 481.658,Z 209.484,A -85,B 0,C 180,E1 -6992.165,E2 -6992.165} C_VEL
LIN {X 0,Y 481.675,Z 209.483,A -85,B 0,C 180,E1 -6994.967,E2 -6994.967} C_VEL
LIN {X 0,Y 481.613,Z 209.492,A -85,B 0,C 180,E1 -6997.703,E2 -6997.703} C_VEL
LIN {X 0,Y 481.658,Z 209.483,A -85,B 0,C 180,E1 -7000.391,E2 -7000.391} C_VEL
LIN {X 0,Y 481.648,Z 209.489,A -85,B 0,C 180,E1 -7003.032,E2 -7003.032} C_VEL
LIN {X 0,Y 481.637,Z 209.488,A -85,B 0,C 180,E1 -7005.637,E2 -7005.637} C_VEL
LIN {X 0,Y 481.745,Z 209.472,A -85,B 0,C 180,E1 -7008.215,E2 -7008.215} C_VEL
LIN {X 0,Y 481.711,Z 209.478,A -85,B 0,C 180,E1 -7011.61,E2 -7011.61} C_VEL
LIN {X 0,Y 481.753,Z 209.471,A -85,B 0,C 180,E1 -7014.139,E2 -7014.139} C_VEL
LIN {X 0,Y 481.873,Z 209.458,A -85,B 0,C 180,E1 -7017.492,E2 -7017.492} C_VEL
LIN {X 0,Y 481.872,Z 209.464,A -85,B 0,C 180,E1 -7020.835,E2 -7020.835} C_VEL
LIN {X 0,Y 481.874,Z 209.459,A -85,B 0,C 180,E1 -7022.507,E2 -7022.507} C_VEL
LIN {X 0,Y 481.783,Z 209.467,A -85,B 0,C 180,E1 -7025.861,E2 -7025.861} C_VEL
LIN {X 0,Y 481.713,Z 209.479,A -85,B 0,C 180,E1 -7028.389,E2 -7028.389} C_VEL
LIN {X 0,Y 481.746,Z 209.472,A -85,B 0,C 180,E1 -7031.785,E2 -7031.785} C_VEL
LIN {X 0,Y 481.693,Z 209.48,A -85,B 0,C 180,E1 -7035.225,E2 -7035.225} C_VEL
LIN {X 0,Y 481.665,Z 209.488,A -85,B 0,C 180,E1 -7038.723,E2 -7038.723} C_VEL
LIN {X 0,Y 481.649,Z 209.484,A -85,B 0,C 180,E1 -7041.394,E2 -7041.394} C_VEL
LIN {X 0,Y 481.648,Z 209.488,A -85,B 0,C 180,E1 -7044.114,E2 -7044.114} C_VEL
LIN {X 0,Y 481.708,Z 209.477,A -85,B 0,C 180,E1 -7047.143,E2 -7047.143} C_VEL
LIN {X 0,Y 481.646,Z 209.486,A -85,B 0,C 180,E1 -7049.743,E2 -7049.743} C_VEL
LIN {X 0,Y 481.633,Z 209.489,A -85,B 0,C 180,E1 -7052.677,E2 -7052.677} C_VEL
LIN {X 0,Y 481.605,Z 209.491,A -85,B 0,C 180,E1 -7055.712,E2 -7055.712} C_VEL
LIN {X 0,Y 481.693,Z 209.479,A -85,B 0,C 180,E1 -7059.358,E2 -7059.358} C_VEL
LIN {X 0,Y 481.644,Z 209.493,A -85,B 0,C 180,E1 -7062.161,E2 -7062.161} C_VEL
LIN {X 0,Y 481.63,Z 209.49,A -85,B 0,C 180,E1 -7064.46,E2 -7064.46} C_VEL
LIN {X 0,Y 481.622,Z 209.493,A -85,B 0,C 180,E1 -7067.842,E2 -7067.842} C_VEL
LIN {X 0,Y 481.691,Z 209.479,A -85,B 0,C 180,E1 -7070.649,E2 -7070.649} C_VEL
LIN {X 0,Y 481.622,Z 209.49,A -85,B 0,C 180,E1 -7074.294,E2 -7074.294} C_VEL
LIN {X 0,Y 481.656,Z 209.485,A -85,B 0,C 180,E1 -7077.329,E2 -7077.329} C_VEL
LIN {X 0,Y 481.672,Z 209.483,A -85,B 0,C 180,E1 -7080.262,E2 -7080.262} C_VEL
LIN {X 0,Y 481.74,Z 209.474,A -85,B 0,C 180,E1 -7083.115,E2 -7083.115} C_VEL
LIN {X 0,Y 481.667,Z 209.487,A -85,B 0,C 180,E1 -7085.889,E2 -7085.889} C_VEL
LIN {X 0,Y 481.628,Z 209.49,A -85,B 0,C 180,E1 -7088.03,E2 -7088.03} C_VEL
LIN {X 0,Y 480.962,Z 209.57,A -85,B 0,C 180,E1 -7088.728,E2 -7088.728} C_VEL
LIN {X 0,Y 478.132,Z 209.927,A -85,B 0,C 180,E1 -7089.862,E2 -7089.862} C_VEL
LIN {X 0,Y 475.747,Z 210.225,A -85,B 0,C 180,E1 -7090.776,E2 -7090.776} C_VEL
LIN {X 0,Y 474.728,Z 210.353,A -85,B 0,C 180,E1 -7091.482,E2 -7091.482} C_VEL
LIN {X 0,Y 474.648,Z 210.36,A -85,B 0,C 180,E1 -7091.721,E2 -7091.721} C_VEL
LIN {X 0,Y 474.695,Z 210.35,A -85,B 0,C 180,E1 -7094.546,E2 -7094.546} C_VEL
LIN {X 0,Y 474.701,Z 210.351,A -85,B 0,C 180,E1 -7098.039,E2 -7098.039} C_VEL
LIN {X 0,Y 474.726,Z 210.353,A -85,B 0,C 180,E1 -7101.487,E2 -7101.487} C_VEL
LIN {X 0,Y 474.769,Z 210.342,A -85,B 0,C 180,E1 -7104.053,E2 -7104.053} C_VEL
LIN {X 0,Y 474.893,Z 210.331,A -85,B 0,C 180,E1 -7107.456,E2 -7107.456} C_VEL
LIN {X 0,Y 474.91,Z 210.324,A -85,B 0,C 180,E1 -7110,E2 -7110} C_VEL
LIN {X 0,Y 474.893,Z 210.327,A -85,B 0,C 180,E1 -7112.544,E2 -7112.544} C_VEL
LIN {X 0,Y 474.764,Z 210.342,A -85,B 0,C 180,E1 -7115.947,E2 -7115.947} C_VEL
LIN {X 0,Y 474.726,Z 210.348,A -85,B 0,C 180,E1 -7118.513,E2 -7118.513} C_VEL
LIN {X 0,Y 474.701,Z 210.349,A -85,B 0,C 180,E1 -7121.961,E2 -7121.961} C_VEL
LIN {X 0,Y 474.695,Z 210.352,A -85,B 0,C 180,E1 -7125.454,E2 -7125.454} C_VEL
LIN {X 0,Y 474.659,Z 210.361,A -85,B 0,C 180,E1 -7129.008,E2 -7129.008} C_VEL
LIN {X 0,Y 474.581,Z 210.364,A -85,B 0,C 180,E1 -7131.727,E2 -7131.727} C_VEL
LIN {X 0,Y 474.649,Z 210.361,A -85,B 0,C 180,E1 -7134.491,E2 -7134.491} C_VEL
LIN {X 0,Y 474.687,Z 210.355,A -85,B 0,C 180,E1 -7137.336,E2 -7137.336} C_VEL
LIN {X 0,Y 474.732,Z 210.465,A -85,B 0,C 180,E1 -7140.126,E2 -7140.126} C_VEL
LIN {X 0,Y 475.603,Z 216.317,A -85,B 0,C 180,E1 -7141.388,E2 -7141.388} C_VEL
LIN {X 0,Y 475.449,Z 225.957,A -85,B 0,C 180,E1 -7143.342,E2 -7143.342} C_VEL
LIN {X 0,Y 478.04,Z 238.958,A -85,B 0,C 180,E1 -7143.643,E2 -7143.643} C_VEL
LIN {X 0,Y 477.279,Z 333.292,A -85,B 0,C 180,E1 -7145.142,E2 -7145.142} C_VEL
LIN {X 0,Y 476.978,Z 346.469,A -85,B 0,C 180,E1 -7145.523,E2 -7145.523} C_VEL
LIN {X 0,Y 476.759,Z 358.468,A -85,B 0,C 180,E1 -7146.036,E2 -7146.036} C_VEL
LIN {X 0,Y 476.363,Z 369.923,A -85,B 0,C 180,E1 -7146.687,E2 -7146.687} C_VEL
LIN {X 0,Y 475.914,Z 381.308,A -85,B 0,C 180,E1 -7147.524,E2 -7147.524} C_VEL
LIN {X 0,Y 475.484,Z 391.971,A -85,B 0,C 180,E1 -7148.504,E2 -7148.504} C_VEL
LIN {X 0,Y 475.067,Z 400.774,A -85,B 0,C 180,E1 -7149.499,E2 -7149.499} C_VEL
LIN {X 0,Y 474.759,Z 409.018,A -85,B 0,C 180,E1 -7150.638,E2 -7150.638} C_VEL
LIN {X 0,Y 474.324,Z 416.996,A -85,B 0,C 180,E1 -7152.003,E2 -7152.003} C_VEL
LIN {X 0,Y 474.14,Z 423.54,A -85,B 0,C 180,E1 -7153.423,E2 -7153.423} C_VEL
LIN {X 0,Y 473.994,Z 427.872,A -85,B 0,C 180,E1 -7154.627,E2 -7154.627} C_VEL
LIN {X 0,Y 473.869,Z 431.175,A -85,B 0,C 180,E1 -7155.809,E2 -7155.809} C_VEL
LIN {X 0,Y 473.781,Z 433.59,A -85,B 0,C 180,E1 -7156.972,E2 -7156.972} C_VEL
LIN {X 0,Y 473.729,Z 435.218,A -85,B 0,C 180,E1 -7158.119,E2 -7158.119} C_VEL
LIN {X 0,Y 473.71,Z 436.088,A -85,B 0,C 180,E1 -7159.248,E2 -7159.248} C_VEL
LIN {X 0,Y 473.642,Z 436.224,A -85,B 0,C 180,E1 -7160.489,E2 -7160.489} C_VEL
LIN {X 0,Y 473.652,Z 435.414,A -85,B 0,C 180,E1 -7161.843,E2 -7161.843} C_VEL
LIN {X 0,Y 473.741,Z 433.528,A -85,B 0,C 180,E1 -7163.226,E2 -7163.226} C_VEL
LIN {X 0,Y 473.857,Z 430.407,A -85,B 0,C 180,E1 -7164.66,E2 -7164.66} C_VEL
LIN {X 0,Y 473.997,Z 425.878,A -85,B 0,C 180,E1 -7166.122,E2 -7166.122} C_VEL
LIN {X 0,Y 474.292,Z 419.633,A -85,B 0,C 180,E1 -7167.621,E2 -7167.621} C_VEL
LIN {X 0,Y 474.615,Z 412.222,A -85,B 0,C 180,E1 -7169.01,E2 -7169.01} C_VEL
LIN {X 0,Y 475.052,Z 403.543,A -85,B 0,C 180,E1 -7170.291,E2 -7170.291} C_VEL
LIN {X 0,Y 475.433,Z 394.223,A -85,B 0,C 180,E1 -7171.408,E2 -7171.408} C_VEL
LIN {X 0,Y 475.84,Z 384.167,A -85,B 0,C 180,E1 -7172.385,E2 -7172.385} C_VEL
LIN {X 0,Y 476.339,Z 372.854,A -85,B 0,C 180,E1 -7173.256,E2 -7173.256} C_VEL
LIN {X 0,Y 476.751,Z 361.625,A -85,B 0,C 180,E1 -7173.938,E2 -7173.938} C_VEL
LIN {X 0,Y 477.109,Z 349.128,A -85,B 0,C 180,E1 -7174.513,E2 -7174.513} C_VEL
LIN {X 0,Y 477.32,Z 337.019,A -85,B 0,C 180,E1 -7174.898,E2 -7174.898} C_VEL
LIN {X 0,Y 477.473,Z 318.398,A -85,B 0,C 180,E1 -7175.241,E2 -7175.241} C_VEL
LIN {X 0,Y 478.231,Z 239.294,A -85,B 0,C 180,E1 -7176.493,E2 -7176.493} C_VEL
LIN {X 0,Y 475.473,Z 225.806,A -85,B 0,C 180,E1 -7176.825,E2 -7176.825} C_VEL
LIN {X 0,Y 475.504,Z 215.341,A -85,B 0,C 180,E1 -7178.751,E2 -7178.751} C_VEL
LIN {X 0,Y 474.669,Z 210.362,A -85,B 0,C 180,E1 -7179.724,E2 -7179.724} C_VEL
LIN {X 0,Y 474.613,Z 210.365,A -85,B 0,C 180,E1 -7182.773,E2 -7182.773} C_VEL
LIN {X 0,Y 474.604,Z 210.372,A -85,B 0,C 180,E1 -7185.42,E2 -7185.42} C_VEL
LIN {X 0,Y 474.69,Z 210.357,A -85,B 0,C 180,E1 -7188.038,E2 -7188.038} C_VEL
LIN {X 0,Y 474.679,Z 210.359,A -85,B 0,C 180,E1 -7191.486,E2 -7191.486} C_VEL
LIN {X 0,Y 474.746,Z 210.346,A -85,B 0,C 180,E1 -7194.052,E2 -7194.052} C_VEL
LIN {X 0,Y 474.842,Z 210.338,A -85,B 0,C 180,E1 -7197.455,E2 -7197.455} C_VEL
LIN {X 0,Y 474.805,Z 210.343,A -85,B 0,C 180,E1 -7200.848,E2 -7200.848} C_VEL
LIN {X 0,Y 474.84,Z 210.336,A -85,B 0,C 180,E1 -7202.545,E2 -7202.545} C_VEL
LIN {X 0,Y 474.717,Z 210.347,A -85,B 0,C 180,E1 -7205.949,E2 -7205.949} C_VEL
LIN {X 0,Y 474.678,Z 210.356,A -85,B 0,C 180,E1 -7208.515,E2 -7208.515} C_VEL
LIN {X 0,Y 474.69,Z 210.35,A -85,B 0,C 180,E1 -7211.963,E2 -7211.963} C_VEL
LIN {X 0,Y 474.654,Z 210.356,A -85,B 0,C 180,E1 -7215.778,E2 -7215.778} C_VEL
LIN {X 0,Y 474.619,Z 210.364,A -85,B 0,C 180,E1 -7219.012,E2 -7219.012} C_VEL
LIN {X 0,Y 474.552,Z 210.369,A -85,B 0,C 180,E1 -7221.731,E2 -7221.731} C_VEL
LIN {X 0,Y 474.618,Z 210.364,A -85,B 0,C 180,E1 -7224.495,E2 -7224.495} C_VEL
LIN {X 0,Y 474.64,Z 210.358,A -85,B 0,C 180,E1 -7227.337,E2 -7227.337} C_VEL
LIN {X 0,Y 474.566,Z 210.371,A -85,B 0,C 180,E1 -7230.813,E2 -7230.813} C_VEL
LIN {X 0,Y 474.604,Z 210.365,A -85,B 0,C 180,E1 -7233.987,E2 -7233.987} C_VEL
LIN {X 0,Y 474.541,Z 210.372,A -85,B 0,C 180,E1 -7236.903,E2 -7236.903} C_VEL
LIN {X 0,Y 474.587,Z 210.366,A -85,B 0,C 180,E1 -7239.649,E2 -7239.649} C_VEL
LIN {X 0,Y 474.596,Z 210.37,A -85,B 0,C 180,E1 -7242.24,E2 -7242.24} C_VEL
LIN {X 0,Y 474.592,Z 210.363,A -85,B 0,C 180,E1 -7245.301,E2 -7245.301} C_VEL
LIN {X 0,Y 474.599,Z 210.369,A -85,B 0,C 180,E1 -7248.218,E2 -7248.218} C_VEL
LIN {X 0,Y 474.624,Z 210.364,A -85,B 0,C 180,E1 -7250.457,E2 -7250.457} C_VEL
LIN {X 0,Y 474.575,Z 210.37,A -85,B 0,C 180,E1 -7253.68,E2 -7253.68} C_VEL
LIN {X 0,Y 474.629,Z 210.361,A -85,B 0,C 180,E1 -7256.783,E2 -7256.783} C_VEL
LIN {X 0,Y 474.594,Z 210.371,A -85,B 0,C 180,E1 -7259.773,E2 -7259.773} C_VEL
LIN {X 0,Y 474.689,Z 210.356,A -85,B 0,C 180,E1 -7262.683,E2 -7262.683} C_VEL
LIN {X 0,Y 474.7,Z 210.566,A -85,B 0,C 180,E1 -7264.038,E2 -7264.038} C_VEL
LIN {X 0,Y 476.662,Z 221.167,A -85,B 0,C 180,E1 -7265.912,E2 -7265.912} C_VEL
LIN {X 0,Y 476.171,Z 237.153,A -85,B 0,C 180,E1 -7268.529,E2 -7268.529} C_VEL
LIN {X 0,Y 475.499,Z 256.782,A -85,B 0,C 180,E1 -7271.702,E2 -7271.702} C_VEL
LIN {X 0,Y 475.243,Z 266.193,A -85,B 0,C 180,E1 -7273.204,E2 -7273.204} C_VEL
LIN {X 0,Y 477.982,Z 285.944,A -85,B 0,C 180,E1 -7273.628,E2 -7273.628} C_VEL
LIN {X 0,Y 477.229,Z 375.858,A -85,B 0,C 180,E1 -7275.067,E2 -7275.067} C_VEL
LIN {X 0,Y 476.916,Z 388.027,A -85,B 0,C 180,E1 -7275.412,E2 -7275.412} C_VEL
LIN {X 0,Y 476.449,Z 400.257,A -85,B 0,C 180,E1 -7275.915,E2 -7275.915} C_VEL
LIN {X 0,Y 476.014,Z 411.811,A -85,B 0,C 180,E1 -7276.555,E2 -7276.555} C_VEL
LIN {X 0,Y 475.596,Z 423.497,A -85,B 0,C 180,E1 -7277.396,E2 -7277.396} C_VEL
LIN {X 0,Y 475.121,Z 434.337,A -85,B 0,C 180,E1 -7278.374,E2 -7278.374} C_VEL
LIN {X 0,Y 474.699,Z 443.05,A -85,B 0,C 180,E1 -7279.336,E2 -7279.336} C_VEL
LIN {X 0,Y 474.397,Z 451.091,A -85,B 0,C 180,E1 -7280.407,E2 -7280.407} C_VEL
LIN {X 0,Y 474.098,Z 458.96,A -85,B 0,C 180,E1 -7281.691,E2 -7281.691} C_VEL
LIN {X 0,Y 473.896,Z 466.195,A -85,B 0,C 180,E1 -7283.187,E2 -7283.187} C_VEL
LIN {X 0,Y 473.833,Z 471.02,A -85,B 0,C 180,E1 -7284.468,E2 -7284.468} C_VEL
LIN {X 0,Y 473.747,Z 474.709,A -85,B 0,C 180,E1 -7285.747,E2 -7285.747} C_VEL
LIN {X 0,Y 473.801,Z 476.619,A -85,B 0,C 180,E1 -7286.599,E2 -7286.599} C_VEL
LIN {X 0,Y 473.762,Z 478.05,A -85,B 0,C 180,E1 -7287.45,E2 -7287.45} C_VEL
LIN {X 0,Y 473.756,Z 479.074,A -85,B 0,C 180,E1 -7288.3,E2 -7288.3} C_VEL
LIN {X 0,Y 473.693,Z 479.702,A -85,B 0,C 180,E1 -7289.15,E2 -7289.15} C_VEL
LIN {X 0,Y 473.679,Z 479.931,A -85,B 0,C 180,E1 -7290,E2 -7290} C_VEL
LIN {X 0,Y 473.756,Z 479.114,A -85,B 0,C 180,E1 -7291.7,E2 -7291.7} C_VEL
LIN {X 0,Y 473.761,Z 478.111,A -85,B 0,C 180,E1 -7292.55,E2 -7292.55} C_VEL
LIN {X 0,Y 473.796,Z 476.695,A -85,B 0,C 180,E1 -7293.401,E2 -7293.401} C_VEL
LIN {X 0,Y 473.761,Z 473.719,A -85,B 0,C 180,E1 -7294.679,E2 -7294.679} C_VEL
LIN {X 0,Y 473.823,Z 469.686,A -85,B 0,C 180,E1 -7295.959,E2 -7295.959} C_VEL
LIN {X 0,Y 473.999,Z 463.471,A -85,B 0,C 180,E1 -7297.453,E2 -7297.453} C_VEL
LIN {X 0,Y 474.212,Z 456.688,A -85,B 0,C 180,E1 -7298.736,E2 -7298.736} C_VEL
LIN {X 0,Y 474.468,Z 448.262,A -85,B 0,C 180,E1 -7300.022,E2 -7300.022} C_VEL
LIN {X 0,Y 474.894,Z 439.586,A -85,B 0,C 180,E1 -7301.091,E2 -7301.091} C_VEL
LIN {X 0,Y 475.331,Z 429.225,A -85,B 0,C 180,E1 -7302.131,E2 -7302.131} C_VEL
LIN {X 0,Y 475.802,Z 418.58,A -85,B 0,C 180,E1 -7302.994,E2 -7302.994} C_VEL
LIN {X 0,Y 476.231,Z 406.517,A -85,B 0,C 180,E1 -7303.765,E2 -7303.765} C_VEL
LIN {X 0,Y 476.661,Z 394.306,A -85,B 0,C 180,E1 -7304.351,E2 -7304.351} C_VEL
LIN {X 0,Y 477.063,Z 381.02,A -85,B 0,C 180,E1 -7304.802,E2 -7304.802} C_VEL
LIN {X 0,Y 477.343,Z 366.23,A -85,B 0,C 180,E1 -7305.093,E2 -7305.093} C_VEL
LIN {X 0,Y 477.789,Z 284.31,A -85,B 0,C 180,E1 -7306.379,E2 -7306.379} C_VEL
LIN {X 0,Y 475.267,Z 266.997,A -85,B 0,C 180,E1 -7306.758,E2 -7306.758} C_VEL
LIN {X 0,Y 475.908,Z 248.261,A -85,B 0,C 180,E1 -7309.853,E2 -7309.853} C_VEL
LIN {X 0,Y 476.637,Z 230.809,A -85,B 0,C 180,E1 -7312.769,E2 -7312.769} C_VEL
LIN {X 0,Y 476.997,Z 222.788,A -85,B 0,C 180,E1 -7314.123,E2 -7314.123} C_VEL
LIN {X 0,Y 474.942,Z 211.685,A -85,B 0,C 180,E1 -7316.147,E2 -7316.147} C_VEL
LIN {X 0,Y 474.684,Z 210.359,A -85,B 0,C 180,E1 -7316.426,E2 -7316.426} C_VEL
LIN {X 0,Y 474.609,Z 210.365,A -85,B 0,C 180,E1 -7319.249,E2 -7319.249} C_VEL
LIN {X 0,Y 474.601,Z 210.366,A -85,B 0,C 180,E1 -7322.427,E2 -7322.427} C_VEL
LIN {X 0,Y 474.602,Z 210.364,A -85,B 0,C 180,E1 -7325.466,E2 -7325.466} C_VEL
LIN {X 0,Y 474.592,Z 210.365,A -85,B 0,C 180,E1 -7328.454,E2 -7328.454} C_VEL
LIN {X 0,Y 474.606,Z 210.361,A -85,B 0,C 180,E1 -7330.956,E2 -7330.956} C_VEL
LIN {X 0,Y 474.583,Z 210.369,A -85,B 0,C 180,E1 -7334.102,E2 -7334.102} C_VEL
LIN {X 0,Y 474.587,Z 210.364,A -85,B 0,C 180,E1 -7337.062,E2 -7337.062} C_VEL
LIN {X 0,Y 474.586,Z 210.365,A -85,B 0,C 180,E1 -7340.351,E2 -7340.351} C_VEL
LIN {X 0,Y 474.558,Z 210.375,A -85,B 0,C 180,E1 -7343.673,E2 -7343.673} C_VEL
LIN {X 0,Y 474.607,Z 210.362,A -85,B 0,C 180,E1 -7346.777,E2 -7346.777} C_VEL
LIN {X 0,Y 474.565,Z 210.371,A -85,B 0,C 180,E1 -7349.767,E2 -7349.767} C_VEL
LIN {X 0,Y 474.657,Z 210.355,A -85,B 0,C 180,E1 -7352.677,E2 -7352.677} C_VEL
LIN {X 0,Y 474.617,Z 210.367,A -85,B 0,C 180,E1 -7355.505,E2 -7355.505} C_VEL
LIN {X 0,Y 474.625,Z 210.365,A -85,B 0,C 180,E1 -7359.183,E2 -7359.183} C_VEL
LIN {X 0,Y 474.61,Z 210.362,A -85,B 0,C 180,E1 -7361.882,E2 -7361.882} C_VEL
LIN {X 0,Y 474.65,Z 210.357,A -85,B 0,C 180,E1 -7364.542,E2 -7364.542} C_VEL
LIN {X 0,Y 474.689,Z 210.351,A -85,B 0,C 180,E1 -7368.037,E2 -7368.037} C_VEL
LIN {X 0,Y 474.677,Z 210.356,A -85,B 0,C 180,E1 -7371.485,E2 -7371.485} C_VEL
LIN {X 0,Y 474.716,Z 210.348,A -85,B 0,C 180,E1 -7374.051,E2 -7374.051} C_VEL
LIN {X 0,Y 474.839,Z 210.335,A -85,B 0,C 180,E1 -7377.455,E2 -7377.455} C_VEL
LIN {X 0,Y 474.823,Z 210.342,A -85,B 0,C 180,E1 -7380.848,E2 -7380.848} C_VEL
LIN {X 0,Y 474.84,Z 210.336,A -85,B 0,C 180,E1 -7382.545,E2 -7382.545} C_VEL
LIN {X 0,Y 474.745,Z 210.344,A -85,B 0,C 180,E1 -7385.948,E2 -7385.948} C_VEL
LIN {X 0,Y 474.678,Z 210.357,A -85,B 0,C 180,E1 -7388.514,E2 -7388.514} C_VEL
LIN {X 0,Y 474.689,Z 210.352,A -85,B 0,C 180,E1 -7391.963,E2 -7391.963} C_VEL
LIN {X 0,Y 474.652,Z 210.356,A -85,B 0,C 180,E1 -7395.778,E2 -7395.778} C_VEL
LIN {X 0,Y 474.62,Z 210.362,A -85,B 0,C 180,E1 -7399.012,E2 -7399.012} C_VEL
LIN {X 0,Y 474.623,Z 210.36,A -85,B 0,C 180,E1 -7401.727,E2 -7401.727} C_VEL
LIN {X 0,Y 474.624,Z 210.367,A -85,B 0,C 180,E1 -7404.494,E2 -7404.494} C_VEL
LIN {X 0,Y 474.657,Z 210.355,A -85,B 0,C 180,E1 -7407.341,E2 -7407.341} C_VEL
LIN {X 0,Y 474.568,Z 210.368,A -85,B 0,C 180,E1 -7410.813,E2 -7410.813} C_VEL
LIN {X 0,Y 474.6,Z 210.366,A -85,B 0,C 180,E1 -7413.987,E2 -7413.987} C_VEL
LIN {X 0,Y 474.539,Z 210.371,A -85,B 0,C 180,E1 -7416.903,E2 -7416.903} C_VEL
LIN {X 0,Y 474.636,Z 210.36,A -85,B 0,C 180,E1 -7419.657,E2 -7419.657} C_VEL
LIN {X 0,Y 474.621,Z 210.36,A -85,B 0,C 180,E1 -7422.933,E2 -7422.933} C_VEL
LIN {X 0,Y 474.581,Z 210.371,A -85,B 0,C 180,E1 -7425.898,E2 -7425.898} C_VEL
LIN {X 0,Y 474.616,Z 210.36,A -85,B 0,C 180,E1 -7429.042,E2 -7429.042} C_VEL
LIN {X 0,Y 474.594,Z 210.368,A -85,B 0,C 180,E1 -7431.706,E2 -7431.706} C_VEL
LIN {X 0,Y 474.61,Z 210.361,A -85,B 0,C 180,E1 -7434.729,E2 -7434.729} C_VEL
LIN {X 0,Y 474.621,Z 210.368,A -85,B 0,C 180,E1 -7437.791,E2 -7437.791} C_VEL
LIN {X 0,Y 474.616,Z 210.36,A -85,B 0,C 180,E1 -7440.886,E2 -7440.886} C_VEL
LIN {X 0,Y 474.655,Z 210.363,A -85,B 0,C 180,E1 -7443.631,E2 -7443.631} C_VEL
LIN {X 0,Y 474.626,Z 210.359,A -85,B 0,C 180,E1 -7446.644,E2 -7446.644} C_VEL
LIN {X 0,Y 474.647,Z 210.358,A -85,B 0,C 180,E1 -7450.092,E2 -7450.092} C_VEL
LIN {X 0,Y 474.648,Z 210.36,A -85,B 0,C 180,E1 -7451.721,E2 -7451.721} C_VEL
LIN {X 0,Y 473.988,Z 210.443,A -85,B 0,C 180,E1 -7452.43,E2 -7452.43} C_VEL
LIN {X 0,Y 471.137,Z 210.801,A -85,B 0,C 180,E1 -7453.581,E2 -7453.581} C_VEL
LIN {X 0,Y 468.72,Z 211.101,A -85,B 0,C 180,E1 -7454.509,E2 -7454.509} C_VEL
LIN {X 0,Y 467.679,Z 211.229,A -85,B 0,C 180,E1 -7455.227,E2 -7455.227} C_VEL
LIN {X 0,Y 467.594,Z 211.237,A -85,B 0,C 180,E1 -7455.47,E2 -7455.47} C_VEL
LIN {X 0,Y 467.65,Z 211.229,A -85,B 0,C 180,E1 -7458.735,E2 -7458.735} C_VEL
LIN {X 0,Y 467.747,Z 211.216,A -85,B 0,C 180,E1 -7462.229,E2 -7462.229} C_VEL
LIN {X 0,Y 467.721,Z 211.221,A -85,B 0,C 180,E1 -7464.828,E2 -7464.828} C_VEL
LIN {X 0,Y 467.858,Z 211.208,A -85,B 0,C 180,E1 -7467.417,E2 -7467.417} C_VEL
LIN {X 0,Y 467.881,Z 211.199,A -85,B 0,C 180,E1 -7470,E2 -7470} C_VEL
LIN {X 0,Y 467.859,Z 211.203,A -85,B 0,C 180,E1 -7472.583,E2 -7472.583} C_VEL
LIN {X 0,Y 467.727,Z 211.218,A -85,B 0,C 180,E1 -7476.037,E2 -7476.037} C_VEL
LIN {X 0,Y 467.679,Z 211.227,A -85,B 0,C 180,E1 -7478.642,E2 -7478.642} C_VEL
LIN {X 0,Y 467.652,Z 211.228,A -85,B 0,C 180,E1 -7482.144,E2 -7482.144} C_VEL
LIN {X 0,Y 467.634,Z 211.23,A -85,B 0,C 180,E1 -7485.693,E2 -7485.693} C_VEL
LIN {X 0,Y 467.611,Z 211.24,A -85,B 0,C 180,E1 -7488.763,E2 -7488.763} C_VEL
LIN {X 0,Y 467.573,Z 211.24,A -85,B 0,C 180,E1 -7491.266,E2 -7491.266} C_VEL
LIN {X 0,Y 467.563,Z 211.239,A -85,B 0,C 180,E1 -7493.941,E2 -7493.941} C_VEL
LIN {X 0,Y 467.616,Z 211.24,A -85,B 0,C 180,E1 -7496.797,E2 -7496.797} C_VEL
LIN {X 0,Y 467.672,Z 211.373,A -85,B 0,C 180,E1 -7499.974,E2 -7499.974} C_VEL
LIN {X 0,Y 468.608,Z 217.217,A -85,B 0,C 180,E1 -7501.256,E2 -7501.256} C_VEL
LIN {X 0,Y 468.462,Z 226.193,A -85,B 0,C 180,E1 -7503.095,E2 -7503.095} C_VEL
LIN {X 0,Y 471.256,Z 240.277,A -85,B 0,C 180,E1 -7503.427,E2 -7503.427} C_VEL
LIN {X 0,Y 470.398,Z 333.449,A -85,B 0,C 180,E1 -7504.93,E2 -7504.93} C_VEL
LIN {X 0,Y 470.086,Z 347.077,A -85,B 0,C 180,E1 -7505.332,E2 -7505.332} C_VEL
LIN {X 0,Y 469.856,Z 359.026,A -85,B 0,C 180,E1 -7505.854,E2 -7505.854} C_VEL
LIN {X 0,Y 469.438,Z 370.287,A -85,B 0,C 180,E1 -7506.506,E2 -7506.506} C_VEL
